LIN {X 0,Y 424.031,Z 1043.321,A -85,B 0,C 180,E1 17866.114,E2 17866.114} C_VEL
LIN {X 0,Y 429.572,Z 1017.595,A -85,B 0,C 180,E1 17864.912,E2 17864.912} C_VEL
LIN {X 0,Y 434.388,Z 990.898,A -85,B 0,C 180,E1 17863.916,E2 17863.916} C_VEL
LIN {X 0,Y 437.982,Z 968.501,A -85,B 0,C 180,E1 17863.251,E2 17863.251} C_VEL
LIN {X 0,Y 429.123,Z 944.994,A -85,B 0,C 180,E1 17861.421,E2 17861.421} C_VEL
LIN {X 0,Y 422.762,Z 922.814,A -85,B 0,C 180,E1 17859.852,E2 17859.852} C_VEL
LIN {X 0,Y 420.084,Z 910.607,A -85,B 0,C 180,E1 17859.018,E2 17859.018} C_VEL
LIN {X 0,Y 421.88,Z 885.683,A -85,B 0,C 180,E1 17856.084,E2 17856.084} C_VEL
LIN {X 0,Y 431.541,Z 834.064,A -85,B 0,C 180,E1 17850.471,E2 17850.471} C_VEL
LIN {X 0,Y 438.469,Z 800.811,A -85,B 0,C 180,E1 17846.841,E2 17846.841} C_VEL
LIN {X 0,Y 442.301,Z 782.261,A -85,B 0,C 180,E1 17844.794,E2 17844.794} C_VEL
LIN {X 0,Y 435.827,Z 764.916,A -85,B 0,C 180,E1 17841.394,E2 17841.394} C_VEL
LIN {X 0,Y 429.102,Z 747.913,A -85,B 0,C 180,E1 17837.774,E2 17837.774} C_VEL
LIN {X 0,Y 422.737,Z 732.697,A -85,B 0,C 180,E1 17834.24,E2 17834.24} C_VEL
LIN {X 0,Y 416.328,Z 717.877,A -85,B 0,C 180,E1 17830.517,E2 17830.517} C_VEL
LIN {X 0,Y 410.081,Z 704.024,A -85,B 0,C 180,E1 17826.721,E2 17826.721} C_VEL
LIN {X 0,Y 404.039,Z 691.12,A -85,B 0,C 180,E1 17822.837,E2 17822.837} C_VEL
LIN {X 0,Y 398.039,Z 678.56,A -85,B 0,C 180,E1 17818.703,E2 17818.703} C_VEL
LIN {X 0,Y 393.112,Z 668.867,A -85,B 0,C 180,E1 17815.185,E2 17815.185} C_VEL
LIN {X 0,Y 390.535,Z 663.891,A -85,B 0,C 180,E1 17813.236,E2 17813.236} C_VEL
LIN {X 0,Y 388.243,Z 659.415,A -85,B 0,C 180,E1 17811.46,E2 17811.46} C_VEL
LIN {X 0,Y 385.936,Z 654.857,A -85,B 0,C 180,E1 17809.551,E2 17809.551} C_VEL
LIN {X 0,Y 384.023,Z 650.756,A -85,B 0,C 180,E1 17807.825,E2 17807.825} C_VEL
LIN {X 0,Y 381.793,Z 647.102,A -85,B 0,C 180,E1 17806.058,E2 17806.058} C_VEL
LIN {X 0,Y 381.224,Z 645.556,A -85,B 0,C 180,E1 17805.416,E2 17805.416} C_VEL
LIN {X 0,Y 379.173,Z 642.261,A -85,B 0,C 180,E1 17803.704,E2 17803.704} C_VEL
LIN {X 0,Y 378.841,Z 640.776,A -85,B 0,C 180,E1 17803.122,E2 17803.122} C_VEL
LIN {X 0,Y 378.842,Z 640.781,A -85,B 0,C 180,E1 17799.111,E2 17799.111} C_VEL
LIN {X 0,Y 378.854,Z 640.787,A -85,B 0,C 180,E1 17795.021,E2 17795.021} C_VEL
LIN {X 0,Y 378.842,Z 640.792,A -85,B 0,C 180,E1 17790.876,E2 17790.876} C_VEL
LIN {X 0,Y 378.847,Z 640.79,A -85,B 0,C 180,E1 17786.784,E2 17786.784} C_VEL
LIN {X 0,Y 378.847,Z 640.785,A -85,B 0,C 180,E1 17782.597,E2 17782.597} C_VEL
LIN {X 0,Y 378.846,Z 640.811,A -85,B 0,C 180,E1 17781.666,E2 17781.666} C_VEL
LIN {X 0,Y 379.93,Z 643.909,A -85,B 0,C 180,E1 17781.165,E2 17781.165} C_VEL
LIN {X 0,Y 381.356,Z 646.05,A -85,B 0,C 180,E1 17780.713,E2 17780.713} C_VEL
LIN {X 0,Y 389.692,Z 662.721,A -85,B 0,C 180,E1 17777.759,E2 17777.759} C_VEL
LIN {X 0,Y 397.273,Z 679.963,A -85,B 0,C 180,E1 17774.988,E2 17774.988} C_VEL
LIN {X 0,Y 404.151,Z 697.993,A -85,B 0,C 180,E1 17772.395,E2 17772.395} C_VEL
LIN {X 0,Y 410.209,Z 717.323,A -85,B 0,C 180,E1 17769.841,E2 17769.841} C_VEL
LIN {X 0,Y 411.164,Z 721.42,A -85,B 0,C 180,E1 17769.346,E2 17769.346} C_VEL
LIN {X 0,Y 407.057,Z 767.944,A -85,B 0,C 180,E1 17765.427,E2 17765.427} C_VEL
LIN {X 0,Y 402.868,Z 818.065,A -85,B 0,C 180,E1 17761.244,E2 17761.244} C_VEL
LIN {X 0,Y 399.655,Z 864.554,A -85,B 0,C 180,E1 17757.511,E2 17757.511} C_VEL
LIN {X 0,Y 400.168,Z 872.112,A -85,B 0,C 180,E1 17757.318,E2 17757.318} C_VEL
LIN {X 0,Y 395.871,Z 1029.252,A -85,B 0,C 180,E1 17754.503,E2 17754.503} C_VEL
LIN {X 0,Y 395.432,Z 1046.821,A -85,B 0,C 180,E1 17754.006,E2 17754.006} C_VEL
LIN {X 0,Y 394.481,Z 1064.239,A -85,B 0,C 180,E1 17753.238,E2 17753.238} C_VEL
LIN {X 0,Y 393.16,Z 1080.267,A -85,B 0,C 180,E1 17752.265,E2 17752.265} C_VEL
LIN {X 0,Y 391.555,Z 1095.097,A -85,B 0,C 180,E1 17751.102,E2 17751.102} C_VEL
LIN {X 0,Y 389.588,Z 1109.913,A -85,B 0,C 180,E1 17749.623,E2 17749.623} C_VEL
LIN {X 0,Y 387.45,Z 1123.854,A -85,B 0,C 180,E1 17747.882,E2 17747.882} C_VEL
LIN {X 0,Y 385.351,Z 1136.244,A -85,B 0,C 180,E1 17745.962,E2 17745.962} C_VEL
LIN {X 0,Y 383.385,Z 1146.973,A -85,B 0,C 180,E1 17743.881,E2 17743.881} C_VEL
LIN {X 0,Y 381.545,Z 1156.777,A -85,B 0,C 180,E1 17741.486,E2 17741.486} C_VEL
LIN {X 0,Y 380.127,Z 1164.442,A -85,B 0,C 180,E1 17739.078,E2 17739.078} C_VEL
LIN {X 0,Y 379.044,Z 1170.475,A -85,B 0,C 180,E1 17736.511,E2 17736.511} C_VEL
LIN {X 0,Y 378.313,Z 1174.865,A -85,B 0,C 180,E1 17733.786,E2 17733.786} C_VEL
LIN {X 0,Y 377.955,Z 1177.371,A -85,B 0,C 180,E1 17731.059,E2 17731.059} C_VEL
LIN {X 0,Y 377.889,Z 1177.992,A -85,B 0,C 180,E1 17728.33,E2 17728.33} C_VEL
LIN {X 0,Y 378.121,Z 1176.838,A -85,B 0,C 180,E1 17725.6,E2 17725.6} C_VEL
LIN {X 0,Y 378.654,Z 1174.068,A -85,B 0,C 180,E1 17723.021,E2 17723.021} C_VEL
LIN {X 0,Y 379.541,Z 1169.524,A -85,B 0,C 180,E1 17720.444,E2 17720.444} C_VEL
LIN {X 0,Y 380.842,Z 1163.047,A -85,B 0,C 180,E1 17717.874,E2 17717.874} C_VEL
LIN {X 0,Y 382.502,Z 1155.002,A -85,B 0,C 180,E1 17715.464,E2 17715.464} C_VEL
LIN {X 0,Y 384.456,Z 1145.382,A -85,B 0,C 180,E1 17713.219,E2 17713.219} C_VEL
LIN {X 0,Y 386.621,Z 1134.139,A -85,B 0,C 180,E1 17711.137,E2 17711.137} C_VEL
LIN {X 0,Y 388.821,Z 1121.791,A -85,B 0,C 180,E1 17709.291,E2 17709.291} C_VEL
LIN {X 0,Y 390.958,Z 1108.464,A -85,B 0,C 180,E1 17707.677,E2 17707.677} C_VEL
LIN {X 0,Y 392.904,Z 1094.157,A -85,B 0,C 180,E1 17706.289,E2 17706.289} C_VEL
LIN {X 0,Y 394.624,Z 1078.729,A -85,B 0,C 180,E1 17705.107,E2 17705.107} C_VEL
LIN {X 0,Y 396.012,Z 1062.182,A -85,B 0,C 180,E1 17704.138,E2 17704.138} C_VEL
LIN {X 0,Y 396.937,Z 1045.139,A -85,B 0,C 180,E1 17703.42,E2 17703.42} C_VEL
LIN {X 0,Y 397.335,Z 1026.569,A -85,B 0,C 180,E1 17702.932,E2 17702.932} C_VEL
LIN {X 0,Y 399.086,Z 959.214,A -85,B 0,C 180,E1 17701.717,E2 17701.717} C_VEL
LIN {X 0,Y 398.467,Z 951.603,A -85,B 0,C 180,E1 17701.515,E2 17701.515} C_VEL
LIN {X 0,Y 393.586,Z 931.664,A -85,B 0,C 180,E1 17700.717,E2 17700.717} C_VEL
LIN {X 0,Y 393.131,Z 925.124,A -85,B 0,C 180,E1 17700.545,E2 17700.545} C_VEL
LIN {X 0,Y 394.72,Z 870.182,A -85,B 0,C 180,E1 17699.543,E2 17699.543} C_VEL
LIN {X 0,Y 394.254,Z 864.919,A -85,B 0,C 180,E1 17699.35,E2 17699.35} C_VEL
LIN {X 0,Y 397.972,Z 816.503,A -85,B 0,C 180,E1 17695.4,E2 17695.4} C_VEL
LIN {X 0,Y 402.393,Z 767.422,A -85,B 0,C 180,E1 17691.256,E2 17691.256} C_VEL
LIN {X 0,Y 403.838,Z 767.962,A -85,B 0,C 180,E1 17691.029,E2 17691.029} C_VEL
LIN {X 0,Y 406.516,Z 766.956,A -85,B 0,C 180,E1 17690.7,E2 17690.7} C_VEL
LIN {X 0,Y 410.432,Z 763.169,A -85,B 0,C 180,E1 17690.312,E2 17690.312} C_VEL
LIN {X 0,Y 412.105,Z 761.138,A -85,B 0,C 180,E1 17690.166,E2 17690.166} C_VEL
LIN {X 0,Y 416.175,Z 759.299,A -85,B 0,C 180,E1 17689.691,E2 17689.691} C_VEL
LIN {X 0,Y 420.888,Z 755.05,A -85,B 0,C 180,E1 17689.229,E2 17689.229} C_VEL
LIN {X 0,Y 422.259,Z 753.761,A -85,B 0,C 180,E1 17689.098,E2 17689.098} C_VEL
LIN {X 0,Y 427.431,Z 750.639,A -85,B 0,C 180,E1 17688.544,E2 17688.544} C_VEL
LIN {X 0,Y 432.452,Z 746.166,A -85,B 0,C 180,E1 17688.069,E2 17688.069} C_VEL
LIN {X 0,Y 436.101,Z 744.14,A -85,B 0,C 180,E1 17687.682,E2 17687.682} C_VEL
LIN {X 0,Y 439.705,Z 749.984,A -85,B 0,C 180,E1 17687.032,E2 17687.032} C_VEL
LIN {X 0,Y 418.06,Z 971.327,A -85,B 0,C 180,E1 17681.624,E2 17681.624} C_VEL
LIN {X 0,Y 415.617,Z 998.063,A -85,B 0,C 180,E1 17680.799,E2 17680.799} C_VEL
LIN {X 0,Y 412.746,Z 1021.843,A -85,B 0,C 180,E1 17679.809,E2 17679.809} C_VEL
LIN {X 0,Y 409.391,Z 1044.41,A -85,B 0,C 180,E1 17678.611,E2 17678.611} C_VEL
LIN {X 0,Y 405.663,Z 1065.433,A -85,B 0,C 180,E1 17677.235,E2 17677.235} C_VEL
LIN {X 0,Y 401.608,Z 1085.727,A -85,B 0,C 180,E1 17675.633,E2 17675.633} C_VEL
LIN {X 0,Y 397.135,Z 1106.048,A -85,B 0,C 180,E1 17673.726,E2 17673.726} C_VEL
LIN {X 0,Y 392.712,Z 1124.842,A -85,B 0,C 180,E1 17671.635,E2 17671.635} C_VEL
LIN {X 0,Y 388.261,Z 1142.534,A -85,B 0,C 180,E1 17669.295,E2 17669.295} C_VEL
LIN {X 0,Y 384.036,Z 1158.977,A -85,B 0,C 180,E1 17666.739,E2 17666.739} C_VEL
LIN {X 0,Y 380.255,Z 1173.722,A -85,B 0,C 180,E1 17664.053,E2 17664.053} C_VEL
LIN {X 0,Y 376.881,Z 1187.211,A -85,B 0,C 180,E1 17661.151,E2 17661.151} C_VEL
LIN {X 0,Y 374.017,Z 1199.238,A -85,B 0,C 180,E1 17658.066,E2 17658.066} C_VEL
LIN {X 0,Y 371.664,Z 1210.327,A -85,B 0,C 180,E1 17654.649,E2 17654.649} C_VEL
LIN {X 0,Y 370.099,Z 1219.053,A -85,B 0,C 180,E1 17651.375,E2 17651.375} C_VEL
LIN {X 0,Y 369.107,Z 1225.945,A -85,B 0,C 180,E1 17648.098,E2 17648.098} C_VEL
LIN {X 0,Y 368.542,Z 1231.531,A -85,B 0,C 180,E1 17644.669,E2 17644.669} C_VEL
LIN {X 0,Y 368.34,Z 1235.206,A -85,B 0,C 180,E1 17641.556,E2 17641.556} C_VEL
LIN {X 0,Y 368.303,Z 1237.705,A -85,B 0,C 180,E1 17638.133,E2 17638.133} C_VEL
LIN {X 0,Y 368.395,Z 1238.777,A -85,B 0,C 180,E1 17634.861,E2 17634.861} C_VEL
LIN {X 0,Y 368.66,Z 1238.351,A -85,B 0,C 180,E1 17631.578,E2 17631.578} C_VEL
LIN {X 0,Y 369.274,Z 1236.414,A -85,B 0,C 180,E1 17627.966,E2 17627.966} C_VEL
LIN {X 0,Y 370.42,Z 1233.083,A -85,B 0,C 180,E1 17624.5,E2 17624.5} C_VEL
LIN {X 0,Y 372.464,Z 1227.596,A -85,B 0,C 180,E1 17620.719,E2 17620.719} C_VEL
LIN {X 0,Y 375.327,Z 1220.672,A -85,B 0,C 180,E1 17617.188,E2 17617.188} C_VEL
LIN {X 0,Y 379.199,Z 1211.964,A -85,B 0,C 180,E1 17613.705,E2 17613.705} C_VEL
LIN {X 0,Y 384.057,Z 1201.512,A -85,B 0,C 180,E1 17610.352,E2 17610.352} C_VEL
LIN {X 0,Y 389.426,Z 1190.172,A -85,B 0,C 180,E1 17607.371,E2 17607.371} C_VEL
LIN {X 0,Y 395.743,Z 1176.713,A -85,B 0,C 180,E1 17604.448,E2 17604.448} C_VEL
LIN {X 0,Y 402.539,Z 1161.94,A -85,B 0,C 180,E1 17601.793,E2 17601.793} C_VEL
LIN {X 0,Y 409.684,Z 1145.817,A -85,B 0,C 180,E1 17599.381,E2 17599.381} C_VEL
LIN {X 0,Y 416.899,Z 1128.807,A -85,B 0,C 180,E1 17597.254,E2 17597.254} C_VEL
LIN {X 0,Y 424.707,Z 1109.687,A -85,B 0,C 180,E1 17595.256,E2 17595.256} C_VEL
LIN {X 0,Y 432.71,Z 1089.815,A -85,B 0,C 180,E1 17593.522,E2 17593.522} C_VEL
LIN {X 0,Y 420.838,Z 1109.322,A -85,B 0,C 180,E1 17591.796,E2 17591.796} C_VEL
LIN {X 0,Y 409.181,Z 1130.653,A -85,B 0,C 180,E1 17589.538,E2 17589.538} C_VEL
LIN {X 0,Y 398.045,Z 1155.339,A -85,B 0,C 180,E1 17586.539,E2 17586.539} C_VEL
LIN {X 0,Y 388.323,Z 1182.093,A -85,B 0,C 180,E1 17582.823,E2 17582.823} C_VEL
LIN {X 0,Y 381.527,Z 1204.921,A -85,B 0,C 180,E1 17579.176,E2 17579.176} C_VEL
LIN {X 0,Y 376.907,Z 1223.133,A -85,B 0,C 180,E1 17575.792,E2 17575.792} C_VEL
LIN {X 0,Y 373.571,Z 1238.131,A -85,B 0,C 180,E1 17572.506,E2 17572.506} C_VEL
LIN {X 0,Y 371.253,Z 1250.21,A -85,B 0,C 180,E1 17569.348,E2 17569.348} C_VEL
LIN {X 0,Y 369.717,Z 1260.007,A -85,B 0,C 180,E1 17566.241,E2 17566.241} C_VEL
LIN {X 0,Y 368.768,Z 1267.805,A -85,B 0,C 180,E1 17563.167,E2 17563.167} C_VEL
LIN {X 0,Y 368.296,Z 1273.929,A -85,B 0,C 180,E1 17560.008,E2 17560.008} C_VEL
LIN {X 0,Y 368.176,Z 1278.219,A -85,B 0,C 180,E1 17556.865,E2 17556.865} C_VEL
LIN {X 0,Y 368.227,Z 1280.634,A -85,B 0,C 180,E1 17553.895,E2 17553.895} C_VEL
LIN {X 0,Y 368.314,Z 1281.463,A -85,B 0,C 180,E1 17550.935,E2 17550.935} C_VEL
LIN {X 0,Y 368.331,Z 1280.72,A -85,B 0,C 180,E1 17547.98,E2 17547.98} C_VEL
LIN {X 0,Y 368.293,Z 1278.415,A -85,B 0,C 180,E1 17545.018,E2 17545.018} C_VEL
LIN {X 0,Y 368.285,Z 1274.288,A -85,B 0,C 180,E1 17541.886,E2 17541.886} C_VEL
LIN {X 0,Y 368.473,Z 1268.454,A -85,B 0,C 180,E1 17538.735,E2 17538.735} C_VEL
LIN {X 0,Y 369.013,Z 1260.875,A -85,B 0,C 180,E1 17535.567,E2 17535.567} C_VEL
LIN {X 0,Y 370.101,Z 1250.861,A -85,B 0,C 180,E1 17532.227,E2 17532.227} C_VEL
LIN {X 0,Y 371.775,Z 1239.387,A -85,B 0,C 180,E1 17529.043,E2 17529.043} C_VEL
LIN {X 0,Y 374.3,Z 1225.03,A -85,B 0,C 180,E1 17525.711,E2 17525.711} C_VEL
LIN {X 0,Y 377.33,Z 1209.895,A -85,B 0,C 180,E1 17522.717,E2 17522.717} C_VEL
LIN {X 0,Y 381.385,Z 1191.503,A -85,B 0,C 180,E1 17519.605,E2 17519.605} C_VEL
LIN {X 0,Y 386.238,Z 1170.811,A -85,B 0,C 180,E1 17516.628,E2 17516.628} C_VEL
LIN {X 0,Y 391.893,Z 1147.584,A -85,B 0,C 180,E1 17513.799,E2 17513.799} C_VEL
LIN {X 0,Y 397.99,Z 1122.971,A -85,B 0,C 180,E1 17511.279,E2 17511.279} C_VEL
LIN {X 0,Y 403.629,Z 1100.15,A -85,B 0,C 180,E1 17509.292,E2 17509.292} C_VEL
LIN {X 0,Y 409.926,Z 1074.472,A -85,B 0,C 180,E1 17507.403,E2 17507.403} C_VEL
LIN {X 0,Y 415.804,Z 1049.73,A -85,B 0,C 180,E1 17505.883,E2 17505.883} C_VEL
LIN {X 0,Y 421.539,Z 1023.87,A -85,B 0,C 180,E1 17504.597,E2 17504.597} C_VEL
LIN {X 0,Y 426.857,Z 997.071,A -85,B 0,C 180,E1 17503.51,E2 17503.51} C_VEL
LIN {X 0,Y 430.603,Z 975.057,A -85,B 0,C 180,E1 17502.8,E2 17502.8} C_VEL
LIN {X 0,Y 431.204,Z 970.753,A -85,B 0,C 180,E1 17502.665,E2 17502.665} C_VEL
LIN {X 0,Y 423.093,Z 948.417,A -85,B 0,C 180,E1 17500.878,E2 17500.878} C_VEL
LIN {X 0,Y 416.791,Z 926.156,A -85,B 0,C 180,E1 17499.286,E2 17499.286} C_VEL
LIN {X 0,Y 413.097,Z 908.739,A -85,B 0,C 180,E1 17498.114,E2 17498.114} C_VEL
LIN {X 0,Y 415.564,Z 883.187,A -85,B 0,C 180,E1 17495.104,E2 17495.104} C_VEL
LIN {X 0,Y 424.795,Z 836.45,A -85,B 0,C 180,E1 17489.985,E2 17489.985} C_VEL
LIN {X 0,Y 431.838,Z 803.495,A -85,B 0,C 180,E1 17486.36,E2 17486.36} C_VEL
LIN {X 0,Y 435.637,Z 785.94,A -85,B 0,C 180,E1 17484.403,E2 17484.403} C_VEL
LIN {X 0,Y 428.843,Z 767.674,A -85,B 0,C 180,E1 17480.757,E2 17480.757} C_VEL
LIN {X 0,Y 422.155,Z 750.724,A -85,B 0,C 180,E1 17477.08,E2 17477.08} C_VEL
LIN {X 0,Y 415.828,Z 735.503,A -85,B 0,C 180,E1 17473.488,E2 17473.488} C_VEL
LIN {X 0,Y 409.667,Z 721.272,A -85,B 0,C 180,E1 17469.837,E2 17469.837} C_VEL
LIN {X 0,Y 403.651,Z 708.035,A -85,B 0,C 180,E1 17466.115,E2 17466.115} C_VEL
LIN {X 0,Y 398.299,Z 696.472,A -85,B 0,C 180,E1 17462.59,E2 17462.59} C_VEL
LIN {X 0,Y 392.484,Z 684.232,A -85,B 0,C 180,E1 17458.54,E2 17458.54} C_VEL
LIN {X 0,Y 387.464,Z 674.344,A -85,B 0,C 180,E1 17454.913,E2 17454.913} C_VEL
LIN {X 0,Y 384.753,Z 669.087,A -85,B 0,C 180,E1 17452.834,E2 17452.834} C_VEL
LIN {X 0,Y 382.847,Z 665.228,A -85,B 0,C 180,E1 17451.287,E2 17451.287} C_VEL
LIN {X 0,Y 380.499,Z 660.623,A -85,B 0,C 180,E1 17449.346,E2 17449.346} C_VEL
LIN {X 0,Y 378.183,Z 656.035,A -85,B 0,C 180,E1 17447.307,E2 17447.307} C_VEL
LIN {X 0,Y 376.218,Z 652.07,A -85,B 0,C 180,E1 17445.533,E2 17445.533} C_VEL
LIN {X 0,Y 373.885,Z 648.166,A -85,B 0,C 180,E1 17443.532,E2 17443.532} C_VEL
LIN {X 0,Y 373.366,Z 646.607,A -85,B 0,C 180,E1 17442.867,E2 17442.867} C_VEL
LIN {X 0,Y 371.234,Z 643.221,A -85,B 0,C 180,E1 17440.968,E2 17440.968} C_VEL
LIN {X 0,Y 370.909,Z 641.765,A -85,B 0,C 180,E1 17440.307,E2 17440.307} C_VEL
LIN {X 0,Y 370.904,Z 641.763,A -85,B 0,C 180,E1 17436.317,E2 17436.317} C_VEL
LIN {X 0,Y 370.921,Z 641.762,A -85,B 0,C 180,E1 17432.146,E2 17432.146} C_VEL
LIN {X 0,Y 370.904,Z 641.769,A -85,B 0,C 180,E1 17427.922,E2 17427.922} C_VEL
LIN {X 0,Y 370.903,Z 641.77,A -85,B 0,C 180,E1 17423.815,E2 17423.815} C_VEL
LIN {X 0,Y 370.931,Z 641.954,A -85,B 0,C 180,E1 17422.896,E2 17422.896} C_VEL
LIN {X 0,Y 371.968,Z 644.859,A -85,B 0,C 180,E1 17422.396,E2 17422.396} C_VEL
LIN {X 0,Y 373.417,Z 646.919,A -85,B 0,C 180,E1 17421.924,E2 17421.924} C_VEL
LIN {X 0,Y 375.245,Z 650.541,A -85,B 0,C 180,E1 17421.23,E2 17421.23} C_VEL
LIN {X 0,Y 382.114,Z 664.007,A -85,B 0,C 180,E1 17418.744,E2 17418.744} C_VEL
LIN {X 0,Y 389.704,Z 680.901,A -85,B 0,C 180,E1 17415.92,E2 17415.92} C_VEL
LIN {X 0,Y 396.49,Z 698.381,A -85,B 0,C 180,E1 17413.306,E2 17413.306} C_VEL
LIN {X 0,Y 402.531,Z 717.046,A -85,B 0,C 180,E1 17410.744,E2 17410.744} C_VEL
LIN {X 0,Y 404.439,Z 724.573,A -85,B 0,C 180,E1 17409.813,E2 17409.813} C_VEL
LIN {X 0,Y 399.978,Z 772.795,A -85,B 0,C 180,E1 17405.709,E2 17405.709} C_VEL
LIN {X 0,Y 395.761,Z 821.856,A -85,B 0,C 180,E1 17401.59,E2 17401.59} C_VEL
LIN {X 0,Y 392.655,Z 865.628,A -85,B 0,C 180,E1 17398.053,E2 17398.053} C_VEL
LIN {X 0,Y 393.135,Z 872.997,A -85,B 0,C 180,E1 17397.862,E2 17397.862} C_VEL
LIN {X 0,Y 388.676,Z 1029.669,A -85,B 0,C 180,E1 17395.01,E2 17395.01} C_VEL
LIN {X 0,Y 388.231,Z 1047.32,A -85,B 0,C 180,E1 17394.51,E2 17394.51} C_VEL
LIN {X 0,Y 387.271,Z 1064.483,A -85,B 0,C 180,E1 17393.749,E2 17393.749} C_VEL
LIN {X 0,Y 385.935,Z 1080.296,A -85,B 0,C 180,E1 17392.786,E2 17392.786} C_VEL
LIN {X 0,Y 384.167,Z 1096.172,A -85,B 0,C 180,E1 17391.527,E2 17391.527} C_VEL
LIN {X 0,Y 382.153,Z 1110.788,A -85,B 0,C 180,E1 17390.042,E2 17390.042} C_VEL
LIN {X 0,Y 379.908,Z 1124.888,A -85,B 0,C 180,E1 17388.25,E2 17388.25} C_VEL
LIN {X 0,Y 377.728,Z 1137.262,A -85,B 0,C 180,E1 17386.293,E2 17386.293} C_VEL
LIN {X 0,Y 375.683,Z 1147.979,A -85,B 0,C 180,E1 17384.171,E2 17384.171} C_VEL
LIN {X 0,Y 373.766,Z 1157.774,A -85,B 0,C 180,E1 17381.728,E2 17381.728} C_VEL
LIN {X 0,Y 372.286,Z 1165.429,A -85,B 0,C 180,E1 17379.271,E2 17379.271} C_VEL
LIN {X 0,Y 371.154,Z 1171.452,A -85,B 0,C 180,E1 17376.65,E2 17376.65} C_VEL
LIN {X 0,Y 370.389,Z 1175.834,A -85,B 0,C 180,E1 17373.868,E2 17373.868} C_VEL
LIN {X 0,Y 370.015,Z 1178.33,A -85,B 0,C 180,E1 17371.082,E2 17371.082} C_VEL
LIN {X 0,Y 369.947,Z 1178.944,A -85,B 0,C 180,E1 17368.294,E2 17368.294} C_VEL
LIN {X 0,Y 370.194,Z 1177.782,A -85,B 0,C 180,E1 17365.505,E2 17365.505} C_VEL
LIN {X 0,Y 370.758,Z 1175.005,A -85,B 0,C 180,E1 17362.872,E2 17362.872} C_VEL
LIN {X 0,Y 371.692,Z 1170.449,A -85,B 0,C 180,E1 17360.241,E2 17360.241} C_VEL
LIN {X 0,Y 373.06,Z 1163.964,A -85,B 0,C 180,E1 17357.617,E2 17357.617} C_VEL
LIN {X 0,Y 374.798,Z 1155.909,A -85,B 0,C 180,E1 17355.159,E2 17355.159} C_VEL
LIN {X 0,Y 376.839,Z 1146.271,A -85,B 0,C 180,E1 17352.869,E2 17352.869} C_VEL
LIN {X 0,Y 379.095,Z 1135.014,A -85,B 0,C 180,E1 17350.748,E2 17350.748} C_VEL
LIN {X 0,Y 381.386,Z 1122.649,A -85,B 0,C 180,E1 17348.868,E2 17348.868} C_VEL
LIN {X 0,Y 383.606,Z 1109.298,A -85,B 0,C 180,E1 17347.226,E2 17347.226} C_VEL
LIN {X 0,Y 385.627,Z 1094.952,A -85,B 0,C 180,E1 17345.814,E2 17345.814} C_VEL
LIN {X 0,Y 387.447,Z 1079.156,A -85,B 0,C 180,E1 17344.589,E2 17344.589} C_VEL
LIN {X 0,Y 388.855,Z 1062.87,A -85,B 0,C 180,E1 17343.626,E2 17343.626} C_VEL
LIN {X 0,Y 389.807,Z 1045.815,A -85,B 0,C 180,E1 17342.9,E2 17342.9} C_VEL
LIN {X 0,Y 390.222,Z 1027.284,A -85,B 0,C 180,E1 17342.408,E2 17342.408} C_VEL
LIN {X 0,Y 393.131,Z 925.124,A -85,B 0,C 180,E1 17340.545,E2 17340.545} C_VEL
LIN {X 0,Y 392.509,Z 917.516,A -85,B 0,C 180,E1 17340.336,E2 17340.336} C_VEL
LIN {X 0,Y 387.765,Z 897.575,A -85,B 0,C 180,E1 17339.513,E2 17339.513} C_VEL
LIN {X 0,Y 387.342,Z 891.036,A -85,B 0,C 180,E1 17339.338,E2 17339.338} C_VEL
LIN {X 0,Y 387.821,Z 871.104,A -85,B 0,C 180,E1 17338.958,E2 17338.958} C_VEL
LIN {X 0,Y 387.337,Z 866.12,A -85,B 0,C 180,E1 17338.785,E2 17338.785} C_VEL
LIN {X 0,Y 391.297,Z 816.823,A -85,B 0,C 180,E1 17334.723,E2 17334.723} C_VEL
LIN {X 0,Y 394.531,Z 781.853,A -85,B 0,C 180,E1 17331.754,E2 17331.754} C_VEL
LIN {X 0,Y 396.413,Z 782.323,A -85,B 0,C 180,E1 17331.461,E2 17331.461} C_VEL
LIN {X 0,Y 399.357,Z 780.833,A -85,B 0,C 180,E1 17331.109,E2 17331.109} C_VEL
LIN {X 0,Y 403.511,Z 776.395,A -85,B 0,C 180,E1 17330.717,E2 17330.717} C_VEL
LIN {X 0,Y 404.367,Z 775.584,A -85,B 0,C 180,E1 17330.633,E2 17330.633} C_VEL
LIN {X 0,Y 408.466,Z 773.667,A -85,B 0,C 180,E1 17330.151,E2 17330.151} C_VEL
LIN {X 0,Y 413.122,Z 769.361,A -85,B 0,C 180,E1 17329.695,E2 17329.695} C_VEL
LIN {X 0,Y 414.607,Z 767.993,A -85,B 0,C 180,E1 17329.552,E2 17329.552} C_VEL
LIN {X 0,Y 419.822,Z 764.787,A -85,B 0,C 180,E1 17328.991,E2 17328.991} C_VEL
LIN {X 0,Y 424.467,Z 760.542,A -85,B 0,C 180,E1 17328.551,E2 17328.551} C_VEL
LIN {X 0,Y 430.338,Z 756.683,A -85,B 0,C 180,E1 17327.951,E2 17327.951} C_VEL
LIN {X 0,Y 433.438,Z 754.075,A -85,B 0,C 180,E1 17327.656,E2 17327.656} C_VEL
LIN {X 0,Y 413.612,Z 946.997,A -85,B 0,C 180,E1 17322.884,E2 17322.884} C_VEL
LIN {X 0,Y 409.476,Z 992.588,A -85,B 0,C 180,E1 17321.596,E2 17321.596} C_VEL
LIN {X 0,Y 406.679,Z 1016.293,A -85,B 0,C 180,E1 17320.659,E2 17320.659} C_VEL
LIN {X 0,Y 403.374,Z 1038.862,A -85,B 0,C 180,E1 17319.507,E2 17319.507} C_VEL
LIN {X 0,Y 399.41,Z 1061.529,A -85,B 0,C 180,E1 17318.074,E2 17318.074} C_VEL
LIN {X 0,Y 395.281,Z 1082.349,A -85,B 0,C 180,E1 17316.474,E2 17316.474} C_VEL
LIN {X 0,Y 390.795,Z 1102.55,A -85,B 0,C 180,E1 17314.612,E2 17314.612} C_VEL
LIN {X 0,Y 386.307,Z 1121.144,A -85,B 0,C 180,E1 17312.573,E2 17312.573} C_VEL
LIN {X 0,Y 381.549,Z 1139.942,A -85,B 0,C 180,E1 17310.138,E2 17310.138} C_VEL
LIN {X 0,Y 377.256,Z 1156.35,A -85,B 0,C 180,E1 17307.634,E2 17307.634} C_VEL
LIN {X 0,Y 373.215,Z 1171.649,A -85,B 0,C 180,E1 17304.874,E2 17304.874} C_VEL
LIN {X 0,Y 369.615,Z 1185.489,A -85,B 0,C 180,E1 17301.921,E2 17301.921} C_VEL
LIN {X 0,Y 366.564,Z 1197.932,A -85,B 0,C 180,E1 17298.776,E2 17298.776} C_VEL
LIN {X 0,Y 364.224,Z 1208.457,A -85,B 0,C 180,E1 17295.607,E2 17295.607} C_VEL
LIN {X 0,Y 362.449,Z 1217.529,A -85,B 0,C 180,E1 17292.264,E2 17292.264} C_VEL
LIN {X 0,Y 361.27,Z 1225.221,A -85,B 0,C 180,E1 17288.756,E2 17288.756} C_VEL
LIN {X 0,Y 360.643,Z 1230.954,A -85,B 0,C 180,E1 17285.409,E2 17285.409} C_VEL
LIN {X 0,Y 360.364,Z 1235.075,A -85,B 0,C 180,E1 17282.067,E2 17282.067} C_VEL
LIN {X 0,Y 360.314,Z 1237.87,A -85,B 0,C 180,E1 17278.728,E2 17278.728} C_VEL
LIN {X 0,Y 360.381,Z 1239.171,A -85,B 0,C 180,E1 17275.385,E2 17275.385} C_VEL
LIN {X 0,Y 360.668,Z 1239.116,A -85,B 0,C 180,E1 17271.786,E2 17271.786} C_VEL
LIN {X 0,Y 361.274,Z 1237.568,A -85,B 0,C 180,E1 17268.182,E2 17268.182} C_VEL
LIN {X 0,Y 362.489,Z 1234.288,A -85,B 0,C 180,E1 17264.481,E2 17264.481} C_VEL
LIN {X 0,Y 364.507,Z 1229.362,A -85,B 0,C 180,E1 17260.781,E2 17260.781} C_VEL
LIN {X 0,Y 367.673,Z 1222.387,A -85,B 0,C 180,E1 17256.945,E2 17256.945} C_VEL
LIN {X 0,Y 371.633,Z 1214.229,A -85,B 0,C 180,E1 17253.472,E2 17253.472} C_VEL
LIN {X 0,Y 376.446,Z 1204.749,A -85,B 0,C 180,E1 17250.218,E2 17250.218} C_VEL
LIN {X 0,Y 382.577,Z 1192.764,A -85,B 0,C 180,E1 17246.891,E2 17246.891} C_VEL
LIN {X 0,Y 389.495,Z 1179.159,A -85,B 0,C 180,E1 17243.811,E2 17243.811} C_VEL
LIN {X 0,Y 397.083,Z 1163.924,A -85,B 0,C 180,E1 17240.985,E2 17240.985} C_VEL
LIN {X 0,Y 404.743,Z 1148.035,A -85,B 0,C 180,E1 17238.541,E2 17238.541} C_VEL
LIN {X 0,Y 413,Z 1130.334,A -85,B 0,C 180,E1 17236.274,E2 17236.274} C_VEL
LIN {X 0,Y 422.364,Z 1109.922,A -85,B 0,C 180,E1 17234.109,E2 17234.109} C_VEL
LIN {X 0,Y 424.839,Z 1104.283,A -85,B 0,C 180,E1 17233.553,E2 17233.553} C_VEL
LIN {X 0,Y 412.217,Z 1123.286,A -85,B 0,C 180,E1 17231.655,E2 17231.655} C_VEL
LIN {X 0,Y 400.152,Z 1143.996,A -85,B 0,C 180,E1 17229.214,E2 17229.214} C_VEL
LIN {X 0,Y 388.536,Z 1168.241,A -85,B 0,C 180,E1 17225.929,E2 17225.929} C_VEL
LIN {X 0,Y 378.618,Z 1194.364,A -85,B 0,C 180,E1 17221.884,E2 17221.884} C_VEL
LIN {X 0,Y 372.234,Z 1214.763,A -85,B 0,C 180,E1 17218.216,E2 17218.216} C_VEL
LIN {X 0,Y 367.836,Z 1231.23,A -85,B 0,C 180,E1 17214.749,E2 17214.749} C_VEL
LIN {X 0,Y 364.84,Z 1244.153,A -85,B 0,C 180,E1 17211.548,E2 17211.548} C_VEL
LIN {X 0,Y 362.608,Z 1255.53,A -85,B 0,C 180,E1 17208.157,E2 17208.157} C_VEL
LIN {X 0,Y 361.241,Z 1264.327,A -85,B 0,C 180,E1 17204.919,E2 17204.919} C_VEL
LIN {X 0,Y 360.491,Z 1271.192,A -85,B 0,C 180,E1 17201.684,E2 17201.684} C_VEL
LIN {X 0,Y 360.205,Z 1276.207,A -85,B 0,C 180,E1 17198.462,E2 17198.462} C_VEL
LIN {X 0,Y 360.196,Z 1279.286,A -85,B 0,C 180,E1 17195.418,E2 17195.418} C_VEL
LIN {X 0,Y 360.287,Z 1280.758,A -85,B 0,C 180,E1 17192.388,E2 17192.388} C_VEL
LIN {X 0,Y 360.355,Z 1280.643,A -85,B 0,C 180,E1 17189.366,E2 17189.366} C_VEL
LIN {X 0,Y 360.336,Z 1278.963,A -85,B 0,C 180,E1 17186.343,E2 17186.343} C_VEL
LIN {X 0,Y 360.298,Z 1275.72,A -85,B 0,C 180,E1 17183.309,E2 17183.309} C_VEL
LIN {X 0,Y 360.383,Z 1270.541,A -85,B 0,C 180,E1 17180.051,E2 17180.051} C_VEL
LIN {X 0,Y 360.749,Z 1263.783,A -85,B 0,C 180,E1 17176.865,E2 17176.865} C_VEL
LIN {X 0,Y 361.575,Z 1255.072,A -85,B 0,C 180,E1 17173.619,E2 17173.619} C_VEL
LIN {X 0,Y 363.068,Z 1243.91,A -85,B 0,C 180,E1 17170.202,E2 17170.202} C_VEL
LIN {X 0,Y 365.236,Z 1230.949,A -85,B 0,C 180,E1 17166.905,E2 17166.905} C_VEL
LIN {X 0,Y 368.172,Z 1215.957,A -85,B 0,C 180,E1 17163.667,E2 17163.667} C_VEL
LIN {X 0,Y 372.108,Z 1197.967,A -85,B 0,C 180,E1 17160.371,E2 17160.371} C_VEL
LIN {X 0,Y 376.898,Z 1177.756,A -85,B 0,C 180,E1 17157.238,E2 17157.238} C_VEL
LIN {X 0,Y 382.202,Z 1156.322,A -85,B 0,C 180,E1 17154.415,E2 17154.415} C_VEL
LIN {X 0,Y 387.725,Z 1134.365,A -85,B 0,C 180,E1 17151.953,E2 17151.953} C_VEL
LIN {X 0,Y 393.451,Z 1112.043,A -85,B 0,C 180,E1 17149.8,E2 17149.8} C_VEL
LIN {X 0,Y 399.741,Z 1087.149,A -85,B 0,C 180,E1 17147.766,E2 17147.766} C_VEL
LIN {X 0,Y 405.799,Z 1062.879,A -85,B 0,C 180,E1 17146.086,E2 17146.086} C_VEL
LIN {X 0,Y 411.795,Z 1037.515,A -85,B 0,C 180,E1 17144.651,E2 17144.651} C_VEL
LIN {X 0,Y 418.027,Z 1009.204,A -85,B 0,C 180,E1 17143.353,E2 17143.353} C_VEL
LIN {X 0,Y 423.019,Z 982.138,A -85,B 0,C 180,E1 17142.347,E2 17142.347} C_VEL
LIN {X 0,Y 424.459,Z 973.014,A -85,B 0,C 180,E1 17142.072,E2 17142.072} C_VEL
LIN {X 0,Y 417.259,Z 952.685,A -85,B 0,C 180,E1 17140.407,E2 17140.407} C_VEL
LIN {X 0,Y 410.942,Z 929.868,A -85,B 0,C 180,E1 17138.728,E2 17138.728} C_VEL
LIN {X 0,Y 406.298,Z 907.138,A -85,B 0,C 180,E1 17137.202,E2 17137.202} C_VEL
LIN {X 0,Y 409.097,Z 882.426,A -85,B 0,C 180,E1 17134.302,E2 17134.302} C_VEL
LIN {X 0,Y 418.081,Z 838.836,A -85,B 0,C 180,E1 17129.483,E2 17129.483} C_VEL
LIN {X 0,Y 425.41,Z 805.389,A -85,B 0,C 180,E1 17125.774,E2 17125.774} C_VEL
LIN {X 0,Y 428.917,Z 789.433,A -85,B 0,C 180,E1 17123.966,E2 17123.966} C_VEL
LIN {X 0,Y 422.062,Z 770.984,A -85,B 0,C 180,E1 17120.236,E2 17120.236} C_VEL
LIN {X 0,Y 415.642,Z 754.638,A -85,B 0,C 180,E1 17116.635,E2 17116.635} C_VEL
LIN {X 0,Y 409.333,Z 739.45,A -85,B 0,C 180,E1 17112.987,E2 17112.987} C_VEL
LIN {X 0,Y 403.446,Z 725.745,A -85,B 0,C 180,E1 17109.414,E2 17109.414} C_VEL
LIN {X 0,Y 397.692,Z 712.969,A -85,B 0,C 180,E1 17105.772,E2 17105.772} C_VEL
LIN {X 0,Y 392.539,Z 701.791,A -85,B 0,C 180,E1 17102.336,E2 17102.336} C_VEL
LIN {X 0,Y 386.923,Z 689.888,A -85,B 0,C 180,E1 17098.371,E2 17098.371} C_VEL
LIN {X 0,Y 381.999,Z 680.08,A -85,B 0,C 180,E1 17094.744,E2 17094.744} C_VEL
LIN {X 0,Y 378.991,Z 674.236,A -85,B 0,C 180,E1 17092.42,E2 17092.42} C_VEL
LIN {X 0,Y 377.459,Z 671.051,A -85,B 0,C 180,E1 17091.125,E2 17091.125} C_VEL
LIN {X 0,Y 374.996,Z 666.28,A -85,B 0,C 180,E1 17089.087,E2 17089.087} C_VEL
LIN {X 0,Y 372.824,Z 661.904,A -85,B 0,C 180,E1 17087.138,E2 17087.138} C_VEL
LIN {X 0,Y 370.455,Z 657.276,A -85,B 0,C 180,E1 17084.983,E2 17084.983} C_VEL
LIN {X 0,Y 368.425,Z 653.503,A -85,B 0,C 180,E1 17083.118,E2 17083.118} C_VEL
LIN {X 0,Y 367.703,Z 652.186,A -85,B 0,C 180,E1 17082.432,E2 17082.432} C_VEL
LIN {X 0,Y 365.814,Z 648.596,A -85,B 0,C 180,E1 17080.552,E2 17080.552} C_VEL
LIN {X 0,Y 365.191,Z 647.358,A -85,B 0,C 180,E1 17079.898,E2 17079.898} C_VEL
LIN {X 0,Y 363.281,Z 644.195,A -85,B 0,C 180,E1 17078.017,E2 17078.017} C_VEL
LIN {X 0,Y 362.965,Z 642.758,A -85,B 0,C 180,E1 17077.315,E2 17077.315} C_VEL
LIN {X 0,Y 362.966,Z 642.751,A -85,B 0,C 180,E1 17073.189,E2 17073.189} C_VEL
LIN {X 0,Y 362.972,Z 642.748,A -85,B 0,C 180,E1 17068.993,E2 17068.993} C_VEL
LIN {X 0,Y 362.962,Z 642.748,A -85,B 0,C 180,E1 17064.847,E2 17064.847} C_VEL
LIN {X 0,Y 362.995,Z 642.975,A -85,B 0,C 180,E1 17064.229,E2 17064.229} C_VEL
LIN {X 0,Y 364.243,Z 646.206,A -85,B 0,C 180,E1 17063.633,E2 17063.633} C_VEL
LIN {X 0,Y 365.577,Z 647.899,A -85,B 0,C 180,E1 17063.202,E2 17063.202} C_VEL
LIN {X 0,Y 367.47,Z 651.68,A -85,B 0,C 180,E1 17062.446,E2 17062.446} C_VEL
LIN {X 0,Y 374.444,Z 665.008,A -85,B 0,C 180,E1 17059.843,E2 17059.843} C_VEL
LIN {X 0,Y 382.472,Z 682.621,A -85,B 0,C 180,E1 17056.769,E2 17056.769} C_VEL
LIN {X 0,Y 389.421,Z 700.31,A -85,B 0,C 180,E1 17054.033,E2 17054.033} C_VEL
LIN {X 0,Y 395.056,Z 717.528,A -85,B 0,C 180,E1 17051.59,E2 17051.59} C_VEL
LIN {X 0,Y 397.699,Z 727.362,A -85,B 0,C 180,E1 17050.309,E2 17050.309} C_VEL
LIN {X 0,Y 393.368,Z 773.02,A -85,B 0,C 180,E1 17046.405,E2 17046.405} C_VEL
LIN {X 0,Y 388.985,Z 822.02,A -85,B 0,C 180,E1 17042.253,E2 17042.253} C_VEL
LIN {X 0,Y 385.685,Z 866.629,A -85,B 0,C 180,E1 17038.617,E2 17038.617} C_VEL
LIN {X 0,Y 386.139,Z 873.877,A -85,B 0,C 180,E1 17038.425,E2 17038.425} C_VEL
LIN {X 0,Y 381.514,Z 1029.966,A -85,B 0,C 180,E1 17035.539,E2 17035.539} C_VEL
LIN {X 0,Y 381.063,Z 1047.819,A -85,B 0,C 180,E1 17035.034,E2 17035.034} C_VEL
LIN {X 0,Y 380.073,Z 1064.989,A -85,B 0,C 180,E1 17034.266,E2 17034.266} C_VEL
LIN {X 0,Y 378.626,Z 1081.516,A -85,B 0,C 180,E1 17033.243,E2 17033.243} C_VEL
LIN {X 0,Y 376.802,Z 1097.246,A -85,B 0,C 180,E1 17031.97,E2 17031.97} C_VEL
LIN {X 0,Y 374.712,Z 1111.837,A -85,B 0,C 180,E1 17030.458,E2 17030.458} C_VEL
LIN {X 0,Y 372.382,Z 1125.922,A -85,B 0,C 180,E1 17028.632,E2 17028.632} C_VEL
LIN {X 0,Y 370.118,Z 1138.28,A -85,B 0,C 180,E1 17026.638,E2 17026.638} C_VEL
LIN {X 0,Y 367.992,Z 1148.984,A -85,B 0,C 180,E1 17024.474,E2 17024.474} C_VEL
LIN {X 0,Y 365.995,Z 1158.771,A -85,B 0,C 180,E1 17021.981,E2 17021.981} C_VEL
LIN {X 0,Y 364.451,Z 1166.415,A -85,B 0,C 180,E1 17019.472,E2 17019.472} C_VEL
LIN {X 0,Y 363.267,Z 1172.429,A -85,B 0,C 180,E1 17016.795,E2 17016.795} C_VEL
LIN {X 0,Y 362.466,Z 1176.803,A -85,B 0,C 180,E1 17013.952,E2 17013.952} C_VEL
LIN {X 0,Y 362.074,Z 1179.289,A -85,B 0,C 180,E1 17011.105,E2 17011.105} C_VEL
LIN {X 0,Y 362.006,Z 1179.895,A -85,B 0,C 180,E1 17008.257,E2 17008.257} C_VEL
LIN {X 0,Y 362.268,Z 1178.726,A -85,B 0,C 180,E1 17005.407,E2 17005.407} C_VEL
LIN {X 0,Y 362.864,Z 1175.943,A -85,B 0,C 180,E1 17002.716,E2 17002.716} C_VEL
LIN {X 0,Y 363.848,Z 1171.375,A -85,B 0,C 180,E1 17000.028,E2 17000.028} C_VEL
LIN {X 0,Y 365.285,Z 1164.88,A -85,B 0,C 180,E1 16997.349,E2 16997.349} C_VEL
LIN {X 0,Y 367.105,Z 1156.815,A -85,B 0,C 180,E1 16994.84,E2 16994.84} C_VEL
LIN {X 0,Y 369.235,Z 1147.16,A -85,B 0,C 180,E1 16992.505,E2 16992.505} C_VEL
LIN {X 0,Y 371.587,Z 1135.889,A -85,B 0,C 180,E1 16990.343,E2 16990.343} C_VEL
LIN {X 0,Y 373.971,Z 1123.506,A -85,B 0,C 180,E1 16988.428,E2 16988.428} C_VEL
LIN {X 0,Y 376.279,Z 1110.13,A -85,B 0,C 180,E1 16986.756,E2 16986.756} C_VEL
LIN {X 0,Y 378.378,Z 1095.747,A -85,B 0,C 180,E1 16985.32,E2 16985.32} C_VEL
LIN {X 0,Y 380.303,Z 1079.578,A -85,B 0,C 180,E1 16984.052,E2 16984.052} C_VEL
LIN {X 0,Y 381.788,Z 1062.851,A -85,B 0,C 180,E1 16983.057,E2 16983.057} C_VEL
LIN {X 0,Y 382.736,Z 1045.741,A -85,B 0,C 180,E1 16982.337,E2 16982.337} C_VEL
LIN {X 0,Y 383.157,Z 1026.651,A -85,B 0,C 180,E1 16981.837,E2 16981.837} C_VEL
LIN {X 0,Y 387.342,Z 891.036,A -85,B 0,C 180,E1 16979.338,E2 16979.338} C_VEL
LIN {X 0,Y 386.699,Z 886.01,A -85,B 0,C 180,E1 16979.174,E2 16979.174} C_VEL
LIN {X 0,Y 381.208,Z 872.033,A -85,B 0,C 180,E1 16978.374,E2 16978.374} C_VEL
LIN {X 0,Y 380.655,Z 869.149,A -85,B 0,C 180,E1 16978.26,E2 16978.26} C_VEL
LIN {X 0,Y 380.54,Z 866.381,A -85,B 0,C 180,E1 16978.118,E2 16978.118} C_VEL
LIN {X 0,Y 384.589,Z 818.117,A -85,B 0,C 180,E1 16974.105,E2 16974.105} C_VEL
LIN {X 0,Y 386.782,Z 796.41,A -85,B 0,C 180,E1 16972.215,E2 16972.215} C_VEL
LIN {X 0,Y 388.899,Z 796.629,A -85,B 0,C 180,E1 16971.897,E2 16971.897} C_VEL
LIN {X 0,Y 392.139,Z 794.633,A -85,B 0,C 180,E1 16971.524,E2 16971.524} C_VEL
LIN {X 0,Y 396.171,Z 790.034,A -85,B 0,C 180,E1 16971.155,E2 16971.155} C_VEL
LIN {X 0,Y 400.261,Z 788.266,A -85,B 0,C 180,E1 16970.66,E2 16970.66} C_VEL
LIN {X 0,Y 404.835,Z 784.257,A -85,B 0,C 180,E1 16970.206,E2 16970.206} C_VEL
LIN {X 0,Y 406.466,Z 782.576,A -85,B 0,C 180,E1 16970.053,E2 16970.053} C_VEL
LIN {X 0,Y 411.49,Z 779.609,A -85,B 0,C 180,E1 16969.501,E2 16969.501} C_VEL
LIN {X 0,Y 417.013,Z 774.661,A -85,B 0,C 180,E1 16968.974,E2 16968.974} C_VEL
LIN {X 0,Y 422.922,Z 770.649,A -85,B 0,C 180,E1 16968.366,E2 16968.366} C_VEL
LIN {X 0,Y 426.136,Z 767.831,A -85,B 0,C 180,E1 16968.065,E2 16968.065} C_VEL
LIN {X 0,Y 406.272,Z 954.541,A -85,B 0,C 180,E1 16963.318,E2 16963.318} C_VEL
LIN {X 0,Y 402.47,Z 994.917,A -85,B 0,C 180,E1 16962.122,E2 16962.122} C_VEL
LIN {X 0,Y 399.678,Z 1017.784,A -85,B 0,C 180,E1 16961.192,E2 16961.192} C_VEL
LIN {X 0,Y 396.339,Z 1039.888,A -85,B 0,C 180,E1 16960.04,E2 16960.04} C_VEL
LIN {X 0,Y 392.21,Z 1062.833,A -85,B 0,C 180,E1 16958.559,E2 16958.559} C_VEL
LIN {X 0,Y 387.922,Z 1083.803,A -85,B 0,C 180,E1 16956.911,E2 16956.911} C_VEL
LIN {X 0,Y 383.292,Z 1104.079,A -85,B 0,C 180,E1 16955,E2 16955} C_VEL
LIN {X 0,Y 378.616,Z 1122.915,A -85,B 0,C 180,E1 16952.878,E2 16952.878} C_VEL
LIN {X 0,Y 373.881,Z 1141.088,A -85,B 0,C 180,E1 16950.462,E2 16950.462} C_VEL
LIN {X 0,Y 369.502,Z 1157.402,A -85,B 0,C 180,E1 16947.914,E2 16947.914} C_VEL
LIN {X 0,Y 365.375,Z 1172.657,A -85,B 0,C 180,E1 16945.099,E2 16945.099} C_VEL
LIN {X 0,Y 361.702,Z 1186.437,A -85,B 0,C 180,E1 16942.084,E2 16942.084} C_VEL
LIN {X 0,Y 358.454,Z 1199.383,A -85,B 0,C 180,E1 16938.711,E2 16938.711} C_VEL
LIN {X 0,Y 356.115,Z 1209.787,A -85,B 0,C 180,E1 16935.47,E2 16935.47} C_VEL
LIN {X 0,Y 354.357,Z 1218.738,A -85,B 0,C 180,E1 16932.052,E2 16932.052} C_VEL
LIN {X 0,Y 353.203,Z 1226.278,A -85,B 0,C 180,E1 16928.465,E2 16928.465} C_VEL
LIN {X 0,Y 352.602,Z 1231.909,A -85,B 0,C 180,E1 16925.043,E2 16925.043} C_VEL
LIN {X 0,Y 352.359,Z 1235.917,A -85,B 0,C 180,E1 16921.626,E2 16921.626} C_VEL
LIN {X 0,Y 352.328,Z 1238.655,A -85,B 0,C 180,E1 16918.048,E2 16918.048} C_VEL
LIN {X 0,Y 352.435,Z 1239.827,A -85,B 0,C 180,E1 16914.774,E2 16914.774} C_VEL
LIN {X 0,Y 352.756,Z 1239.673,A -85,B 0,C 180,E1 16911.195,E2 16911.195} C_VEL
LIN {X 0,Y 353.473,Z 1238.116,A -85,B 0,C 180,E1 16907.585,E2 16907.585} C_VEL
LIN {X 0,Y 354.863,Z 1234.857,A -85,B 0,C 180,E1 16903.802,E2 16903.802} C_VEL
LIN {X 0,Y 357.127,Z 1229.932,A -85,B 0,C 180,E1 16900.027,E2 16900.027} C_VEL
LIN {X 0,Y 360.477,Z 1223.264,A -85,B 0,C 180,E1 16896.259,E2 16896.259} C_VEL
LIN {X 0,Y 364.954,Z 1214.856,A -85,B 0,C 180,E1 16892.587,E2 16892.587} C_VEL
LIN {X 0,Y 370.407,Z 1204.943,A -85,B 0,C 180,E1 16889.142,E2 16889.142} C_VEL
LIN {X 0,Y 376.726,Z 1193.619,A -85,B 0,C 180,E1 16885.942,E2 16885.942} C_VEL
LIN {X 0,Y 384.114,Z 1180.219,A -85,B 0,C 180,E1 16882.849,E2 16882.849} C_VEL
LIN {X 0,Y 392.194,Z 1165.305,A -85,B 0,C 180,E1 16880.024,E2 16880.024} C_VEL
LIN {X 0,Y 400.798,Z 1148.942,A -85,B 0,C 180,E1 16877.462,E2 16877.462} C_VEL
LIN {X 0,Y 410.701,Z 1129.762,A -85,B 0,C 180,E1 16874.988,E2 16874.988} C_VEL
LIN {X 0,Y 417.009,Z 1117.356,A -85,B 0,C 180,E1 16873.616,E2 16873.616} C_VEL
LIN {X 0,Y 403.208,Z 1136.644,A -85,B 0,C 180,E1 16871.463,E2 16871.463} C_VEL
LIN {X 0,Y 391.342,Z 1155.862,A -85,B 0,C 180,E1 16868.944,E2 16868.944} C_VEL
LIN {X 0,Y 380.228,Z 1177.478,A -85,B 0,C 180,E1 16865.72,E2 16865.72} C_VEL
LIN {X 0,Y 370.28,Z 1201.781,A -85,B 0,C 180,E1 16861.594,E2 16861.594} C_VEL
LIN {X 0,Y 363.63,Z 1221.456,A -85,B 0,C 180,E1 16857.693,E2 16857.693} C_VEL
LIN {X 0,Y 359.271,Z 1236.662,A -85,B 0,C 180,E1 16854.151,E2 16854.151} C_VEL
LIN {X 0,Y 356.133,Z 1249.615,A -85,B 0,C 180,E1 16850.548,E2 16850.548} C_VEL
LIN {X 0,Y 354.178,Z 1259.361,A -85,B 0,C 180,E1 16847.245,E2 16847.245} C_VEL
LIN {X 0,Y 352.96,Z 1267.193,A -85,B 0,C 180,E1 16843.935,E2 16843.935} C_VEL
LIN {X 0,Y 352.356,Z 1273.167,A -85,B 0,C 180,E1 16840.631,E2 16840.631} C_VEL
LIN {X 0,Y 352.184,Z 1277.331,A -85,B 0,C 180,E1 16837.342,E2 16837.342} C_VEL
LIN {X 0,Y 352.235,Z 1279.625,A -85,B 0,C 180,E1 16834.235,E2 16834.235} C_VEL
LIN {X 0,Y 352.347,Z 1280.326,A -85,B 0,C 180,E1 16831.14,E2 16831.14} C_VEL
LIN {X 0,Y 352.384,Z 1279.448,A -85,B 0,C 180,E1 16828.051,E2 16828.051} C_VEL
LIN {X 0,Y 352.346,Z 1276.959,A -85,B 0,C 180,E1 16824.922,E2 16824.922} C_VEL
LIN {X 0,Y 352.339,Z 1272.719,A -85,B 0,C 180,E1 16821.681,E2 16821.681} C_VEL
LIN {X 0,Y 352.544,Z 1266.697,A -85,B 0,C 180,E1 16818.385,E2 16818.385} C_VEL
LIN {X 0,Y 353.147,Z 1258.858,A -85,B 0,C 180,E1 16815.072,E2 16815.072} C_VEL
LIN {X 0,Y 354.366,Z 1248.6,A -85,B 0,C 180,E1 16811.58,E2 16811.58} C_VEL
LIN {X 0,Y 356.21,Z 1236.808,A -85,B 0,C 180,E1 16808.255,E2 16808.255} C_VEL
LIN {X 0,Y 358.984,Z 1222.137,A -85,B 0,C 180,E1 16804.779,E2 16804.779} C_VEL
LIN {X 0,Y 362.509,Z 1205.759,A -85,B 0,C 180,E1 16801.502,E2 16801.502} C_VEL
LIN {X 0,Y 366.71,Z 1187.842,A -85,B 0,C 180,E1 16798.435,E2 16798.435} C_VEL
LIN {X 0,Y 371.834,Z 1167.311,A -85,B 0,C 180,E1 16795.434,E2 16795.434} C_VEL
LIN {X 0,Y 377.567,Z 1145.07,A -85,B 0,C 180,E1 16792.67,E2 16792.67} C_VEL
LIN {X 0,Y 384.222,Z 1119.532,A -85,B 0,C 180,E1 16790.003,E2 16790.003} C_VEL
LIN {X 0,Y 390.306,Z 1096.244,A -85,B 0,C 180,E1 16787.943,E2 16787.943} C_VEL
LIN {X 0,Y 396.869,Z 1070.769,A -85,B 0,C 180,E1 16786.047,E2 16786.047} C_VEL
LIN {X 0,Y 403.033,Z 1046.021,A -85,B 0,C 180,E1 16784.503,E2 16784.503} C_VEL
LIN {X 0,Y 409.078,Z 1020.075,A -85,B 0,C 180,E1 16783.199,E2 16783.199} C_VEL
LIN {X 0,Y 414.754,Z 992.319,A -85,B 0,C 180,E1 16782.057,E2 16782.057} C_VEL
LIN {X 0,Y 417.665,Z 975.288,A -85,B 0,C 180,E1 16781.469,E2 16781.469} C_VEL
LIN {X 0,Y 410.847,Z 954.975,A -85,B 0,C 180,E1 16779.772,E2 16779.772} C_VEL
LIN {X 0,Y 404.852,Z 932.686,A -85,B 0,C 180,E1 16778.107,E2 16778.107} C_VEL
LIN {X 0,Y 400.088,Z 908.548,A -85,B 0,C 180,E1 16776.462,E2 16776.462} C_VEL
LIN {X 0,Y 399.547,Z 904.545,A -85,B 0,C 180,E1 16776.2,E2 16776.2} C_VEL
LIN {X 0,Y 403.163,Z 878.968,A -85,B 0,C 180,E1 16773.189,E2 16773.189} C_VEL
LIN {X 0,Y 411.37,Z 840.996,A -85,B 0,C 180,E1 16768.957,E2 16768.957} C_VEL
LIN {X 0,Y 418.905,Z 807.81,A -85,B 0,C 180,E1 16765.231,E2 16765.231} C_VEL
LIN {X 0,Y 422.157,Z 792.892,A -85,B 0,C 180,E1 16763.529,E2 16763.529} C_VEL
LIN {X 0,Y 415.76,Z 775.535,A -85,B 0,C 180,E1 16759.969,E2 16759.969} C_VEL
LIN {X 0,Y 409.608,Z 759.722,A -85,B 0,C 180,E1 16756.449,E2 16756.449} C_VEL
LIN {X 0,Y 403.559,Z 744.998,A -85,B 0,C 180,E1 16752.885,E2 16752.885} C_VEL
LIN {X 0,Y 397.468,Z 730.715,A -85,B 0,C 180,E1 16749.119,E2 16749.119} C_VEL
LIN {X 0,Y 391.913,Z 718.311,A -85,B 0,C 180,E1 16745.564,E2 16745.564} C_VEL
LIN {X 0,Y 386.748,Z 707.066,A -85,B 0,C 180,E1 16742.074,E2 16742.074} C_VEL
LIN {X 0,Y 381.358,Z 695.535,A -85,B 0,C 180,E1 16738.197,E2 16738.197} C_VEL
LIN {X 0,Y 376.456,Z 685.682,A -85,B 0,C 180,E1 16734.513,E2 16734.513} C_VEL
LIN {X 0,Y 372.359,Z 677.296,A -85,B 0,C 180,E1 16731.164,E2 16731.164} C_VEL
LIN {X 0,Y 369.632,Z 672.131,A -85,B 0,C 180,E1 16728.927,E2 16728.927} C_VEL
LIN {X 0,Y 367.428,Z 667.721,A -85,B 0,C 180,E1 16726.946,E2 16726.946} C_VEL
LIN {X 0,Y 364.959,Z 662.944,A -85,B 0,C 180,E1 16724.651,E2 16724.651} C_VEL
LIN {X 0,Y 362.544,Z 658.274,A -85,B 0,C 180,E1 16722.339,E2 16722.339} C_VEL
LIN {X 0,Y 360.588,Z 654.604,A -85,B 0,C 180,E1 16720.395,E2 16720.395} C_VEL
LIN {X 0,Y 359.886,Z 653.292,A -85,B 0,C 180,E1 16719.678,E2 16719.678} C_VEL
LIN {X 0,Y 357.971,Z 649.816,A -85,B 0,C 180,E1 16717.674,E2 16717.674} C_VEL
LIN {X 0,Y 357.358,Z 648.461,A -85,B 0,C 180,E1 16716.938,E2 16716.938} C_VEL
LIN {X 0,Y 355.378,Z 645.272,A -85,B 0,C 180,E1 16714.858,E2 16714.858} C_VEL
LIN {X 0,Y 355.028,Z 643.751,A -85,B 0,C 180,E1 16714.117,E2 16714.117} C_VEL
LIN {X 0,Y 355.03,Z 643.745,A -85,B 0,C 180,E1 16710.099,E2 16710.099} C_VEL
LIN {X 0,Y 355.036,Z 643.739,A -85,B 0,C 180,E1 16705.888,E2 16705.888} C_VEL
LIN {X 0,Y 355.062,Z 643.942,A -85,B 0,C 180,E1 16705.67,E2 16705.67} C_VEL
LIN {X 0,Y 356.407,Z 647.33,A -85,B 0,C 180,E1 16704.999,E2 16704.999} C_VEL
LIN {X 0,Y 357.872,Z 649.434,A -85,B 0,C 180,E1 16704.468,E2 16704.468} C_VEL
LIN {X 0,Y 359.803,Z 653.008,A -85,B 0,C 180,E1 16703.693,E2 16703.693} C_VEL
LIN {X 0,Y 365.627,Z 663.999,A -85,B 0,C 180,E1 16701.426,E2 16701.426} C_VEL
LIN {X 0,Y 372.284,Z 677.592,A -85,B 0,C 180,E1 16698.85,E2 16698.85} C_VEL
LIN {X 0,Y 379.567,Z 694.853,A -85,B 0,C 180,E1 16695.936,E2 16695.936} C_VEL
LIN {X 0,Y 385.882,Z 712.44,A -85,B 0,C 180,E1 16693.271,E2 16693.271} C_VEL
LIN {X 0,Y 391.092,Z 730.068,A -85,B 0,C 180,E1 16690.852,E2 16690.852} C_VEL
LIN {X 0,Y 386.345,Z 778.034,A -85,B 0,C 180,E1 16686.713,E2 16686.713} C_VEL
LIN {X 0,Y 381.94,Z 825.838,A -85,B 0,C 180,E1 16682.632,E2 16682.632} C_VEL
LIN {X 0,Y 378.768,Z 867.779,A -85,B 0,C 180,E1 16679.197,E2 16679.197} C_VEL
LIN {X 0,Y 379.181,Z 874.758,A -85,B 0,C 180,E1 16679.009,E2 16679.009} C_VEL
LIN {X 0,Y 374.384,Z 1030.378,A -85,B 0,C 180,E1 16676.086,E2 16676.086} C_VEL
LIN {X 0,Y 373.913,Z 1048.559,A -85,B 0,C 180,E1 16675.568,E2 16675.568} C_VEL
LIN {X 0,Y 372.918,Z 1065.357,A -85,B 0,C 180,E1 16674.81,E2 16674.81} C_VEL
LIN {X 0,Y 371.474,Z 1081.436,A -85,B 0,C 180,E1 16673.81,E2 16673.81} C_VEL
LIN {X 0,Y 369.572,Z 1097.456,A -85,B 0,C 180,E1 16672.509,E2 16672.509} C_VEL
LIN {X 0,Y 367.4,Z 1112.242,A -85,B 0,C 180,E1 16670.968,E2 16670.968} C_VEL
LIN {X 0,Y 365.067,Z 1125.885,A -85,B 0,C 180,E1 16669.186,E2 16669.186} C_VEL
LIN {X 0,Y 362.691,Z 1138.422,A -85,B 0,C 180,E1 16667.154,E2 16667.154} C_VEL
LIN {X 0,Y 360.46,Z 1149.314,A -85,B 0,C 180,E1 16664.948,E2 16664.948} C_VEL
LIN {X 0,Y 358.464,Z 1158.662,A -85,B 0,C 180,E1 16662.564,E2 16662.564} C_VEL
LIN {X 0,Y 356.792,Z 1166.528,A -85,B 0,C 180,E1 16660.004,E2 16660.004} C_VEL
LIN {X 0,Y 355.568,Z 1172.511,A -85,B 0,C 180,E1 16657.43,E2 16657.43} C_VEL
LIN {X 0,Y 354.691,Z 1176.98,A -85,B 0,C 180,E1 16654.687,E2 16654.687} C_VEL
LIN {X 0,Y 354.185,Z 1179.83,A -85,B 0,C 180,E1 16651.777,E2 16651.777} C_VEL
LIN {X 0,Y 354.052,Z 1180.882,A -85,B 0,C 180,E1 16648.865,E2 16648.865} C_VEL
LIN {X 0,Y 354.233,Z 1180.209,A -85,B 0,C 180,E1 16646.113,E2 16646.113} C_VEL
LIN {X 0,Y 354.786,Z 1177.668,A -85,B 0,C 180,E1 16643.2,E2 16643.2} C_VEL
LIN {X 0,Y 355.794,Z 1173.235,A -85,B 0,C 180,E1 16640.29,E2 16640.29} C_VEL
LIN {X 0,Y 357.12,Z 1167.546,A -85,B 0,C 180,E1 16637.712,E2 16637.712} C_VEL
LIN {X 0,Y 358.903,Z 1159.933,A -85,B 0,C 180,E1 16635.147,E2 16635.147} C_VEL
LIN {X 0,Y 361.009,Z 1150.823,A -85,B 0,C 180,E1 16632.759,E2 16632.759} C_VEL
LIN {X 0,Y 363.366,Z 1140.254,A -85,B 0,C 180,E1 16630.549,E2 16630.549} C_VEL
LIN {X 0,Y 365.862,Z 1128.127,A -85,B 0,C 180,E1 16628.515,E2 16628.515} C_VEL
LIN {X 0,Y 368.301,Z 1114.855,A -85,B 0,C 180,E1 16626.731,E2 16626.731} C_VEL
LIN {X 0,Y 370.692,Z 1099.847,A -85,B 0,C 180,E1 16625.114,E2 16625.114} C_VEL
LIN {X 0,Y 372.684,Z 1084.729,A -85,B 0,C 180,E1 16623.828,E2 16623.828} C_VEL
LIN {X 0,Y 374.296,Z 1068.49,A -85,B 0,C 180,E1 16622.774,E2 16622.774} C_VEL
LIN {X 0,Y 375.474,Z 1050.725,A -85,B 0,C 180,E1 16621.935,E2 16621.935} C_VEL
LIN {X 0,Y 376.052,Z 1033.082,A -85,B 0,C 180,E1 16621.394,E2 16621.394} C_VEL
LIN {X 0,Y 378.077,Z 961.199,A -85,B 0,C 180,E1 16620.021,E2 16620.021} C_VEL
LIN {X 0,Y 380.97,Z 872.082,A -85,B 0,C 180,E1 16618.353,E2 16618.353} C_VEL
LIN {X 0,Y 380.655,Z 869.149,A -85,B 0,C 180,E1 16618.26,E2 16618.26} C_VEL
LIN {X 0,Y 381.012,Z 864.008,A -85,B 0,C 180,E1 16617.957,E2 16617.957} C_VEL
LIN {X 0,Y 380.466,Z 858.441,A -85,B 0,C 180,E1 16617.398,E2 16617.398} C_VEL
LIN {X 0,Y 376.153,Z 843.922,A -85,B 0,C 180,E1 16615.593,E2 16615.593} C_VEL
LIN {X 0,Y 376.006,Z 840.131,A -85,B 0,C 180,E1 16615.228,E2 16615.228} C_VEL
LIN {X 0,Y 378.808,Z 810.804,A -85,B 0,C 180,E1 16612.713,E2 16612.713} C_VEL
LIN {X 0,Y 380.541,Z 811.21,A -85,B 0,C 180,E1 16612.438,E2 16612.438} C_VEL
LIN {X 0,Y 383.514,Z 809.733,A -85,B 0,C 180,E1 16612.072,E2 16612.072} C_VEL
LIN {X 0,Y 387.617,Z 805.464,A -85,B 0,C 180,E1 16611.68,E2 16611.68} C_VEL
LIN {X 0,Y 388.636,Z 804.343,A -85,B 0,C 180,E1 16611.584,E2 16611.584} C_VEL
LIN {X 0,Y 392.801,Z 802.349,A -85,B 0,C 180,E1 16611.087,E2 16611.087} C_VEL
LIN {X 0,Y 397.554,Z 797.906,A -85,B 0,C 180,E1 16610.62,E2 16610.62} C_VEL
LIN {X 0,Y 398.626,Z 796.924,A -85,B 0,C 180,E1 16610.514,E2 16610.514} C_VEL
LIN {X 0,Y 403.678,Z 793.948,A -85,B 0,C 180,E1 16609.956,E2 16609.956} C_VEL
LIN {X 0,Y 409.026,Z 789.166,A -85,B 0,C 180,E1 16609.438,E2 16609.438} C_VEL
LIN {X 0,Y 414.994,Z 785.142,A -85,B 0,C 180,E1 16608.823,E2 16608.823} C_VEL
LIN {X 0,Y 418.727,Z 781.834,A -85,B 0,C 180,E1 16608.471,E2 16608.471} C_VEL
LIN {X 0,Y 398.619,Z 965.445,A -85,B 0,C 180,E1 16603.655,E2 16603.655} C_VEL
LIN {X 0,Y 395.393,Z 997.955,A -85,B 0,C 180,E1 16602.633,E2 16602.633} C_VEL
LIN {X 0,Y 392.4,Z 1021.352,A -85,B 0,C 180,E1 16601.64,E2 16601.64} C_VEL
LIN {X 0,Y 388.785,Z 1044.015,A -85,B 0,C 180,E1 16600.399,E2 16600.399} C_VEL
LIN {X 0,Y 384.768,Z 1065.269,A -85,B 0,C 180,E1 16598.968,E2 16598.968} C_VEL
LIN {X 0,Y 380.2,Z 1086.712,A -85,B 0,C 180,E1 16597.22,E2 16597.22} C_VEL
LIN {X 0,Y 375.542,Z 1106.496,A -85,B 0,C 180,E1 16595.294,E2 16595.294} C_VEL
LIN {X 0,Y 370.587,Z 1125.941,A -85,B 0,C 180,E1 16593.026,E2 16593.026} C_VEL
LIN {X 0,Y 365.92,Z 1143.233,A -85,B 0,C 180,E1 16590.639,E2 16590.639} C_VEL
LIN {X 0,Y 361.249,Z 1160.14,A -85,B 0,C 180,E1 16587.89,E2 16587.89} C_VEL
LIN {X 0,Y 357.105,Z 1175.157,A -85,B 0,C 180,E1 16585.012,E2 16585.012} C_VEL
LIN {X 0,Y 353.442,Z 1188.673,A -85,B 0,C 180,E1 16581.927,E2 16581.927} C_VEL
LIN {X 0,Y 350.34,Z 1200.803,A -85,B 0,C 180,E1 16578.635,E2 16578.635} C_VEL
LIN {X 0,Y 347.905,Z 1211.484,A -85,B 0,C 180,E1 16575.161,E2 16575.161} C_VEL
LIN {X 0,Y 346.2,Z 1220.311,A -85,B 0,C 180,E1 16571.664,E2 16571.664} C_VEL
LIN {X 0,Y 345.134,Z 1227.315,A -85,B 0,C 180,E1 16568.161,E2 16568.161} C_VEL
LIN {X 0,Y 344.548,Z 1233.014,A -85,B 0,C 180,E1 16564.494,E2 16564.494} C_VEL
LIN {X 0,Y 344.359,Z 1236.752,A -85,B 0,C 180,E1 16561.165,E2 16561.165} C_VEL
LIN {X 0,Y 344.342,Z 1239.364,A -85,B 0,C 180,E1 16557.504,E2 16557.504} C_VEL
LIN {X 0,Y 344.511,Z 1240.523,A -85,B 0,C 180,E1 16554.003,E2 16554.003} C_VEL
LIN {X 0,Y 344.92,Z 1240.183,A -85,B 0,C 180,E1 16550.32,E2 16550.32} C_VEL
LIN {X 0,Y 345.911,Z 1238.211,A -85,B 0,C 180,E1 16546.289,E2 16546.289} C_VEL
LIN {X 0,Y 347.649,Z 1234.718,A -85,B 0,C 180,E1 16542.422,E2 16542.422} C_VEL
LIN {X 0,Y 350.529,Z 1229.322,A -85,B 0,C 180,E1 16538.409,E2 16538.409} C_VEL
LIN {X 0,Y 354.649,Z 1222.045,A -85,B 0,C 180,E1 16534.446,E2 16534.446} C_VEL
LIN {X 0,Y 360.127,Z 1212.751,A -85,B 0,C 180,E1 16530.565,E2 16530.565} C_VEL
LIN {X 0,Y 366.716,Z 1201.809,A -85,B 0,C 180,E1 16526.953,E2 16526.953} C_VEL
LIN {X 0,Y 374.288,Z 1189.292,A -85,B 0,C 180,E1 16523.625,E2 16523.625} C_VEL
LIN {X 0,Y 382.661,Z 1175.255,A -85,B 0,C 180,E1 16520.583,E2 16520.583} C_VEL
LIN {X 0,Y 391.704,Z 1159.732,A -85,B 0,C 180,E1 16517.828,E2 16517.828} C_VEL
LIN {X 0,Y 401.866,Z 1142.008,A -85,B 0,C 180,E1 16515.24,E2 16515.24} C_VEL
LIN {X 0,Y 409.004,Z 1129.536,A -85,B 0,C 180,E1 16513.682,E2 16513.682} C_VEL
LIN {X 0,Y 395.992,Z 1146.385,A -85,B 0,C 180,E1 16511.614,E2 16511.614} C_VEL
LIN {X 0,Y 383.446,Z 1165.135,A -85,B 0,C 180,E1 16508.937,E2 16508.937} C_VEL
LIN {X 0,Y 371.32,Z 1187.258,A -85,B 0,C 180,E1 16505.321,E2 16505.321} C_VEL
LIN {X 0,Y 361.543,Z 1209.506,A -85,B 0,C 180,E1 16501.145,E2 16501.145} C_VEL
LIN {X 0,Y 355.214,Z 1227.019,A -85,B 0,C 180,E1 16497.314,E2 16497.314} C_VEL
LIN {X 0,Y 350.715,Z 1241.692,A -85,B 0,C 180,E1 16493.526,E2 16493.526} C_VEL
LIN {X 0,Y 347.7,Z 1253.396,A -85,B 0,C 180,E1 16489.887,E2 16489.887} C_VEL
LIN {X 0,Y 345.848,Z 1262.361,A -85,B 0,C 180,E1 16486.461,E2 16486.461} C_VEL
LIN {X 0,Y 344.734,Z 1269.584,A -85,B 0,C 180,E1 16482.951,E2 16482.951} C_VEL
LIN {X 0,Y 344.25,Z 1274.762,A -85,B 0,C 180,E1 16479.532,E2 16479.532} C_VEL
LIN {X 0,Y 344.197,Z 1278.073,A -85,B 0,C 180,E1 16476.173,E2 16476.173} C_VEL
LIN {X 0,Y 344.299,Z 1279.582,A -85,B 0,C 180,E1 16472.999,E2 16472.999} C_VEL
LIN {X 0,Y 344.405,Z 1279.51,A -85,B 0,C 180,E1 16469.836,E2 16469.836} C_VEL
LIN {X 0,Y 344.399,Z 1277.993,A -85,B 0,C 180,E1 16466.84,E2 16466.84} C_VEL
LIN {X 0,Y 344.353,Z 1274.84,A -85,B 0,C 180,E1 16463.667,E2 16463.667} C_VEL
LIN {X 0,Y 344.411,Z 1269.799,A -85,B 0,C 180,E1 16460.309,E2 16460.309} C_VEL
LIN {X 0,Y 344.766,Z 1262.995,A -85,B 0,C 180,E1 16456.928,E2 16456.928} C_VEL
LIN {X 0,Y 345.601,Z 1254.332,A -85,B 0,C 180,E1 16453.531,E2 16453.531} C_VEL
LIN {X 0,Y 347.213,Z 1242.787,A -85,B 0,C 180,E1 16449.852,E2 16449.852} C_VEL
LIN {X 0,Y 349.517,Z 1229.707,A -85,B 0,C 180,E1 16446.393,E2 16446.393} C_VEL
LIN {X 0,Y 352.63,Z 1214.672,A -85,B 0,C 180,E1 16443.023,E2 16443.023} C_VEL
LIN {X 0,Y 356.896,Z 1196.237,A -85,B 0,C 180,E1 16439.533,E2 16439.533} C_VEL
LIN {X 0,Y 361.984,Z 1175.884,A -85,B 0,C 180,E1 16436.278,E2 16436.278} C_VEL
LIN {X 0,Y 367.628,Z 1154.328,A -85,B 0,C 180,E1 16433.356,E2 16433.356} C_VEL
LIN {X 0,Y 373.47,Z 1132.297,A -85,B 0,C 180,E1 16430.817,E2 16430.817} C_VEL
LIN {X 0,Y 379.733,Z 1109.148,A -85,B 0,C 180,E1 16428.533,E2 16428.533} C_VEL
LIN {X 0,Y 386.434,Z 1083.872,A -85,B 0,C 180,E1 16426.427,E2 16426.427} C_VEL
LIN {X 0,Y 392.989,Z 1058.863,A -85,B 0,C 180,E1 16424.676,E2 16424.676} C_VEL
LIN {X 0,Y 399.288,Z 1033.531,A -85,B 0,C 180,E1 16423.225,E2 16423.225} C_VEL
LIN {X 0,Y 405.742,Z 1005.283,A -85,B 0,C 180,E1 16421.911,E2 16421.911} C_VEL
LIN {X 0,Y 410.954,Z 978.508,A -85,B 0,C 180,E1 16420.903,E2 16420.903} C_VEL
LIN {X 0,Y 410.643,Z 976.712,A -85,B 0,C 180,E1 16420.78,E2 16420.78} C_VEL
LIN {X 0,Y 403.376,Z 953.769,A -85,B 0,C 180,E1 16418.851,E2 16418.851} C_VEL
LIN {X 0,Y 397.665,Z 930.392,A -85,B 0,C 180,E1 16417.107,E2 16417.107} C_VEL
LIN {X 0,Y 393.321,Z 905.631,A -85,B 0,C 180,E1 16415.424,E2 16415.424} C_VEL
LIN {X 0,Y 392.987,Z 902.226,A -85,B 0,C 180,E1 16415.19,E2 16415.19} C_VEL
LIN {X 0,Y 397.309,Z 876.15,A -85,B 0,C 180,E1 16412.12,E2 16412.12} C_VEL
LIN {X 0,Y 405.296,Z 840.466,A -85,B 0,C 180,E1 16408.113,E2 16408.113} C_VEL
LIN {X 0,Y 412.887,Z 807.878,A -85,B 0,C 180,E1 16404.424,E2 16404.424} C_VEL
LIN {X 0,Y 415.459,Z 796.446,A -85,B 0,C 180,E1 16403.097,E2 16403.097} C_VEL
LIN {X 0,Y 408.994,Z 778.832,A -85,B 0,C 180,E1 16399.42,E2 16399.42} C_VEL
LIN {X 0,Y 402.665,Z 762.477,A -85,B 0,C 180,E1 16395.704,E2 16395.704} C_VEL
LIN {X 0,Y 396.166,Z 746.705,A -85,B 0,C 180,E1 16391.797,E2 16391.797} C_VEL
LIN {X 0,Y 390.324,Z 733.013,A -85,B 0,C 180,E1 16388.1,E2 16388.1} C_VEL
LIN {X 0,Y 384.594,Z 720.255,A -85,B 0,C 180,E1 16384.324,E2 16384.324} C_VEL
LIN {X 0,Y 379.298,Z 708.729,A -85,B 0,C 180,E1 16380.604,E2 16380.604} C_VEL
LIN {X 0,Y 373.787,Z 696.944,A -85,B 0,C 180,E1 16376.473,E2 16376.473} C_VEL
LIN {X 0,Y 368.922,Z 687.198,A -85,B 0,C 180,E1 16372.681,E2 16372.681} C_VEL
LIN {X 0,Y 366.38,Z 682.213,A -85,B 0,C 180,E1 16370.576,E2 16370.576} C_VEL
LIN {X 0,Y 364.068,Z 677.649,A -85,B 0,C 180,E1 16368.595,E2 16368.595} C_VEL
LIN {X 0,Y 361.816,Z 673.213,A -85,B 0,C 180,E1 16366.577,E2 16366.577} C_VEL
LIN {X 0,Y 359.694,Z 668.917,A -85,B 0,C 180,E1 16364.522,E2 16364.522} C_VEL
LIN {X 0,Y 357.212,Z 664.159,A -85,B 0,C 180,E1 16362.112,E2 16362.112} C_VEL
LIN {X 0,Y 355.255,Z 660.195,A -85,B 0,C 180,E1 16360.054,E2 16360.054} C_VEL
LIN {X 0,Y 352.781,Z 655.831,A -85,B 0,C 180,E1 16357.503,E2 16357.503} C_VEL
LIN {X 0,Y 352.154,Z 654.496,A -85,B 0,C 180,E1 16356.754,E2 16356.754} C_VEL
LIN {X 0,Y 350.202,Z 651.224,A -85,B 0,C 180,E1 16354.642,E2 16354.642} C_VEL
LIN {X 0,Y 349.723,Z 649.735,A -85,B 0,C 180,E1 16353.858,E2 16353.858} C_VEL
LIN {X 0,Y 347.531,Z 646.513,A -85,B 0,C 180,E1 16351.471,E2 16351.471} C_VEL
LIN {X 0,Y 347.094,Z 644.739,A -85,B 0,C 180,E1 16350.451,E2 16350.451} C_VEL
LIN {X 0,Y 347.107,Z 644.851,A -85,B 0,C 180,E1 16347.256,E2 16347.256} C_VEL
LIN {X 0,Y 348.405,Z 648.233,A -85,B 0,C 180,E1 16346.563,E2 16346.563} C_VEL
LIN {X 0,Y 350.058,Z 650.344,A -85,B 0,C 180,E1 16345.955,E2 16345.955} C_VEL
LIN {X 0,Y 351.844,Z 653.864,A -85,B 0,C 180,E1 16345.165,E2 16345.165} C_VEL
LIN {X 0,Y 357.692,Z 664.435,A -85,B 0,C 180,E1 16342.81,E2 16342.81} C_VEL
LIN {X 0,Y 365.019,Z 679.295,A -85,B 0,C 180,E1 16339.837,E2 16339.837} C_VEL
LIN {X 0,Y 372.108,Z 695.702,A -85,B 0,C 180,E1 16336.957,E2 16336.957} C_VEL
LIN {X 0,Y 378.176,Z 712.234,A -85,B 0,C 180,E1 16334.34,E2 16334.34} C_VEL
LIN {X 0,Y 383.801,Z 730.56,A -85,B 0,C 180,E1 16331.72,E2 16331.72} C_VEL
LIN {X 0,Y 384.434,Z 733.56,A -85,B 0,C 180,E1 16331.345,E2 16331.345} C_VEL
LIN {X 0,Y 379.624,Z 780.17,A -85,B 0,C 180,E1 16327.283,E2 16327.283} C_VEL
LIN {X 0,Y 375.024,Z 828.473,A -85,B 0,C 180,E1 16323.129,E2 16323.129} C_VEL
LIN {X 0,Y 371.86,Z 868.639,A -85,B 0,C 180,E1 16319.807,E2 16319.807} C_VEL
LIN {X 0,Y 372.262,Z 875.637,A -85,B 0,C 180,E1 16319.615,E2 16319.615} C_VEL
LIN {X 0,Y 367.289,Z 1030.788,A -85,B 0,C 180,E1 16316.653,E2 16316.653} C_VEL
LIN {X 0,Y 366.803,Z 1049.16,A -85,B 0,C 180,E1 16316.127,E2 16316.127} C_VEL
LIN {X 0,Y 365.797,Z 1065.731,A -85,B 0,C 180,E1 16315.374,E2 16315.374} C_VEL
LIN {X 0,Y 364.233,Z 1082.544,A -85,B 0,C 180,E1 16314.314,E2 16314.314} C_VEL
LIN {X 0,Y 362.256,Z 1098.561,A -85,B 0,C 180,E1 16312.987,E2 16312.987} C_VEL
LIN {X 0,Y 360.005,Z 1113.29,A -85,B 0,C 180,E1 16311.419,E2 16311.419} C_VEL
LIN {X 0,Y 357.584,Z 1126.918,A -85,B 0,C 180,E1 16309.603,E2 16309.603} C_VEL
LIN {X 0,Y 355.117,Z 1139.443,A -85,B 0,C 180,E1 16307.532,E2 16307.532} C_VEL
LIN {X 0,Y 352.796,Z 1150.319,A -85,B 0,C 180,E1 16305.28,E2 16305.28} C_VEL
LIN {X 0,Y 350.688,Z 1159.793,A -85,B 0,C 180,E1 16302.807,E2 16302.807} C_VEL
LIN {X 0,Y 348.973,Z 1167.517,A -85,B 0,C 180,E1 16300.23,E2 16300.23} C_VEL
LIN {X 0,Y 347.694,Z 1173.491,A -85,B 0,C 180,E1 16297.599,E2 16297.599} C_VEL
LIN {X 0,Y 346.776,Z 1177.949,A -85,B 0,C 180,E1 16294.794,E2 16294.794} C_VEL
LIN {X 0,Y 346.248,Z 1180.792,A -85,B 0,C 180,E1 16291.818,E2 16291.818} C_VEL
LIN {X 0,Y 346.109,Z 1181.837,A -85,B 0,C 180,E1 16288.839,E2 16288.839} C_VEL
LIN {X 0,Y 346.302,Z 1181.153,A -85,B 0,C 180,E1 16286.024,E2 16286.024} C_VEL
LIN {X 0,Y 346.887,Z 1178.605,A -85,B 0,C 180,E1 16283.044,E2 16283.044} C_VEL
LIN {X 0,Y 347.949,Z 1174.164,A -85,B 0,C 180,E1 16280.069,E2 16280.069} C_VEL
LIN {X 0,Y 349.354,Z 1168.425,A -85,B 0,C 180,E1 16277.418,E2 16277.418} C_VEL
LIN {X 0,Y 351.21,Z 1160.84,A -85,B 0,C 180,E1 16274.814,E2 16274.814} C_VEL
LIN {X 0,Y 353.412,Z 1151.719,A -85,B 0,C 180,E1 16272.376,E2 16272.376} C_VEL
LIN {X 0,Y 355.868,Z 1141.136,A -85,B 0,C 180,E1 16270.123,E2 16270.123} C_VEL
LIN {X 0,Y 358.465,Z 1128.986,A -85,B 0,C 180,E1 16268.049,E2 16268.049} C_VEL
LIN {X 0,Y 360.979,Z 1115.818,A -85,B 0,C 180,E1 16266.247,E2 16266.247} C_VEL
LIN {X 0,Y 363.348,Z 1101.542,A -85,B 0,C 180,E1 16264.674,E2 16264.674} C_VEL
LIN {X 0,Y 365.456,Z 1086.262,A -85,B 0,C 180,E1 16263.337,E2 16263.337} C_VEL
LIN {X 0,Y 367.166,Z 1069.889,A -85,B 0,C 180,E1 16262.244,E2 16262.244} C_VEL
LIN {X 0,Y 368.39,Z 1052.413,A -85,B 0,C 180,E1 16261.396,E2 16261.396} C_VEL
LIN {X 0,Y 369.023,Z 1034.815,A -85,B 0,C 180,E1 16260.835,E2 16260.835} C_VEL
LIN {X 0,Y 370.73,Z 974.091,A -85,B 0,C 180,E1 16259.645,E2 16259.645} C_VEL
LIN {X 0,Y 374.15,Z 872.934,A -85,B 0,C 180,E1 16257.722,E2 16257.722} C_VEL
LIN {X 0,Y 373.669,Z 868.082,A -85,B 0,C 180,E1 16257.552,E2 16257.552} C_VEL
LIN {X 0,Y 376.006,Z 840.131,A -85,B 0,C 180,E1 16255.228,E2 16255.228} C_VEL
LIN {X 0,Y 375.738,Z 836.309,A -85,B 0,C 180,E1 16254.795,E2 16254.795} C_VEL
LIN {X 0,Y 373.742,Z 829.807,A -85,B 0,C 180,E1 16253.595,E2 16253.595} C_VEL
LIN {X 0,Y 373.936,Z 826.676,A -85,B 0,C 180,E1 16252.948,E2 16252.948} C_VEL
LIN {X 0,Y 375.597,Z 824.285,A -85,B 0,C 180,E1 16252.536,E2 16252.536} C_VEL
LIN {X 0,Y 375.835,Z 824.083,A -85,B 0,C 180,E1 16252.508,E2 16252.508} C_VEL
LIN {X 0,Y 379.777,Z 819.868,A -85,B 0,C 180,E1 16252.137,E2 16252.137} C_VEL
LIN {X 0,Y 380.617,Z 818.824,A -85,B 0,C 180,E1 16252.066,E2 16252.066} C_VEL
LIN {X 0,Y 384.569,Z 817.036,A -85,B 0,C 180,E1 16251.579,E2 16251.579} C_VEL
LIN {X 0,Y 389.245,Z 812.906,A -85,B 0,C 180,E1 16251.11,E2 16251.11} C_VEL
LIN {X 0,Y 391.099,Z 811.137,A -85,B 0,C 180,E1 16250.933,E2 16250.933} C_VEL
LIN {X 0,Y 396.213,Z 807.944,A -85,B 0,C 180,E1 16250.367,E2 16250.367} C_VEL
LIN {X 0,Y 400.786,Z 803.706,A -85,B 0,C 180,E1 16249.933,E2 16249.933} C_VEL
LIN {X 0,Y 406.756,Z 799.82,A -85,B 0,C 180,E1 16249.303,E2 16249.303} C_VEL
LIN {X 0,Y 411.228,Z 795.867,A -85,B 0,C 180,E1 16248.881,E2 16248.881} C_VEL
LIN {X 0,Y 391.33,Z 972.101,A -85,B 0,C 180,E1 16244.113,E2 16244.113} C_VEL
LIN {X 0,Y 388.17,Z 1002.205,A -85,B 0,C 180,E1 16243.104,E2 16243.104} C_VEL
LIN {X 0,Y 385.025,Z 1025.237,A -85,B 0,C 180,E1 16242.068,E2 16242.068} C_VEL
LIN {X 0,Y 381.443,Z 1046.785,A -85,B 0,C 180,E1 16240.846,E2 16240.846} C_VEL
LIN {X 0,Y 377.139,Z 1068.555,A -85,B 0,C 180,E1 16239.32,E2 16239.32} C_VEL
LIN {X 0,Y 372.488,Z 1089.509,A -85,B 0,C 180,E1 16237.543,E2 16237.543} C_VEL
LIN {X 0,Y 367.525,Z 1109.813,A -85,B 0,C 180,E1 16235.481,E2 16235.481} C_VEL
LIN {X 0,Y 362.559,Z 1128.778,A -85,B 0,C 180,E1 16233.192,E2 16233.192} C_VEL
LIN {X 0,Y 357.55,Z 1146.795,A -85,B 0,C 180,E1 16230.595,E2 16230.595} C_VEL
LIN {X 0,Y 352.995,Z 1162.808,A -85,B 0,C 180,E1 16227.864,E2 16227.864} C_VEL
LIN {X 0,Y 348.617,Z 1178.242,A -85,B 0,C 180,E1 16224.756,E2 16224.756} C_VEL
LIN {X 0,Y 344.995,Z 1191.49,A -85,B 0,C 180,E1 16221.597,E2 16221.597} C_VEL
LIN {X 0,Y 341.966,Z 1203.25,A -85,B 0,C 180,E1 16218.232,E2 16218.232} C_VEL
LIN {X 0,Y 339.585,Z 1213.593,A -85,B 0,C 180,E1 16214.668,E2 16214.668} C_VEL
LIN {X 0,Y 337.974,Z 1222.126,A -85,B 0,C 180,E1 16211.087,E2 16211.087} C_VEL
LIN {X 0,Y 336.991,Z 1228.925,A -85,B 0,C 180,E1 16207.502,E2 16207.502} C_VEL
LIN {X 0,Y 336.505,Z 1234.108,A -85,B 0,C 180,E1 16203.919,E2 16203.919} C_VEL
LIN {X 0,Y 336.359,Z 1237.9,A -85,B 0,C 180,E1 16200.341,E2 16200.341} C_VEL
LIN {X 0,Y 336.376,Z 1240.155,A -85,B 0,C 180,E1 16196.762,E2 16196.762} C_VEL
LIN {X 0,Y 336.601,Z 1241.15,A -85,B 0,C 180,E1 16193.004,E2 16193.004} C_VEL
LIN {X 0,Y 337.162,Z 1240.683,A -85,B 0,C 180,E1 16189.232,E2 16189.232} C_VEL
LIN {X 0,Y 338.336,Z 1238.594,A -85,B 0,C 180,E1 16185.276,E2 16185.276} C_VEL
LIN {X 0,Y 340.494,Z 1234.762,A -85,B 0,C 180,E1 16181.154,E2 16181.154} C_VEL
LIN {X 0,Y 343.845,Z 1229.167,A -85,B 0,C 180,E1 16177.066,E2 16177.066} C_VEL
LIN {X 0,Y 348.308,Z 1222.095,A -85,B 0,C 180,E1 16173.211,E2 16173.211} C_VEL
LIN {X 0,Y 354.098,Z 1213.214,A -85,B 0,C 180,E1 16169.451,E2 16169.451} C_VEL
LIN {X 0,Y 361.237,Z 1202.37,A -85,B 0,C 180,E1 16165.813,E2 16165.813} C_VEL
LIN {X 0,Y 369.371,Z 1190.001,A -85,B 0,C 180,E1 16162.477,E2 16162.477} C_VEL
LIN {X 0,Y 378.323,Z 1176.204,A -85,B 0,C 180,E1 16159.446,E2 16159.446} C_VEL
LIN {X 0,Y 388.491,Z 1160.294,A -85,B 0,C 180,E1 16156.591,E2 16156.591} C_VEL
LIN {X 0,Y 399.97,Z 1142.312,A -85,B 0,C 180,E1 16153.947,E2 16153.947} C_VEL
LIN {X 0,Y 400.857,Z 1140.894,A -85,B 0,C 180,E1 16153.756,E2 16153.756} C_VEL
LIN {X 0,Y 387.19,Z 1157.492,A -85,B 0,C 180,E1 16151.504,E2 16151.504} C_VEL
LIN {X 0,Y 374.45,Z 1175.409,A -85,B 0,C 180,E1 16148.673,E2 16148.673} C_VEL
LIN {X 0,Y 361.784,Z 1197.347,A -85,B 0,C 180,E1 16144.706,E2 16144.706} C_VEL
LIN {X 0,Y 351.896,Z 1218.794,A -85,B 0,C 180,E1 16140.196,E2 16140.196} C_VEL
LIN {X 0,Y 345.671,Z 1235.357,A -85,B 0,C 180,E1 16136.085,E2 16136.085} C_VEL
LIN {X 0,Y 341.531,Z 1248.474,A -85,B 0,C 180,E1 16132.192,E2 16132.192} C_VEL
LIN {X 0,Y 338.918,Z 1258.444,A -85,B 0,C 180,E1 16128.582,E2 16128.582} C_VEL
LIN {X 0,Y 337.274,Z 1266.436,A -85,B 0,C 180,E1 16124.949,E2 16124.949} C_VEL
LIN {X 0,Y 336.46,Z 1272.233,A -85,B 0,C 180,E1 16121.487,E2 16121.487} C_VEL
LIN {X 0,Y 336.189,Z 1276.263,A -85,B 0,C 180,E1 16118.038,E2 16118.038} C_VEL
LIN {X 0,Y 336.244,Z 1278.49,A -85,B 0,C 180,E1 16114.778,E2 16114.778} C_VEL
LIN {X 0,Y 336.378,Z 1279.137,A -85,B 0,C 180,E1 16111.535,E2 16111.535} C_VEL
LIN {X 0,Y 336.439,Z 1278.299,A -85,B 0,C 180,E1 16108.47,E2 16108.47} C_VEL
LIN {X 0,Y 336.41,Z 1275.859,A -85,B 0,C 180,E1 16105.229,E2 16105.229} C_VEL
LIN {X 0,Y 336.385,Z 1271.82,A -85,B 0,C 180,E1 16101.972,E2 16101.972} C_VEL
LIN {X 0,Y 336.569,Z 1265.839,A -85,B 0,C 180,E1 16098.521,E2 16098.521} C_VEL
LIN {X 0,Y 337.168,Z 1258.043,A -85,B 0,C 180,E1 16095.051,E2 16095.051} C_VEL
LIN {X 0,Y 338.424,Z 1247.768,A -85,B 0,C 180,E1 16091.395,E2 16091.395} C_VEL
LIN {X 0,Y 340.351,Z 1235.986,A -85,B 0,C 180,E1 16087.914,E2 16087.914} C_VEL
LIN {X 0,Y 343.268,Z 1221.275,A -85,B 0,C 180,E1 16084.28,E2 16084.28} C_VEL
LIN {X 0,Y 346.777,Z 1205.767,A -85,B 0,C 180,E1 16081.029,E2 16081.029} C_VEL
LIN {X 0,Y 351.388,Z 1187.094,A -85,B 0,C 180,E1 16077.686,E2 16077.686} C_VEL
LIN {X 0,Y 356.97,Z 1165.853,A -85,B 0,C 180,E1 16074.467,E2 16074.467} C_VEL
LIN {X 0,Y 363.379,Z 1142.309,A -85,B 0,C 180,E1 16071.462,E2 16071.462} C_VEL
LIN {X 0,Y 370.454,Z 1116.483,A -85,B 0,C 180,E1 16068.709,E2 16068.709} C_VEL
LIN {X 0,Y 377.126,Z 1092.276,A -85,B 0,C 180,E1 16066.53,E2 16066.53} C_VEL
LIN {X 0,Y 384.039,Z 1066.596,A -85,B 0,C 180,E1 16064.599,E2 16064.599} C_VEL
LIN {X 0,Y 390.811,Z 1040.575,A -85,B 0,C 180,E1 16062.972,E2 16062.972} C_VEL
LIN {X 0,Y 397.023,Z 1015.099,A -85,B 0,C 180,E1 16061.685,E2 16061.685} C_VEL
LIN {X 0,Y 402.854,Z 987.238,A -85,B 0,C 180,E1 16060.529,E2 16060.529} C_VEL
LIN {X 0,Y 404.227,Z 979.907,A -85,B 0,C 180,E1 16060.258,E2 16060.258} C_VEL
LIN {X 0,Y 397.133,Z 956.513,A -85,B 0,C 180,E1 16058.229,E2 16058.229} C_VEL
LIN {X 0,Y 391.307,Z 931.725,A -85,B 0,C 180,E1 16056.346,E2 16056.346} C_VEL
LIN {X 0,Y 387.146,Z 906.351,A -85,B 0,C 180,E1 16054.614,E2 16054.614} C_VEL
LIN {X 0,Y 386.509,Z 900.127,A -85,B 0,C 180,E1 16054.196,E2 16054.196} C_VEL
LIN {X 0,Y 391.889,Z 871.612,A -85,B 0,C 180,E1 16050.854,E2 16050.854} C_VEL
LIN {X 0,Y 400.023,Z 836.864,A -85,B 0,C 180,E1 16046.9,E2 16046.9} C_VEL
LIN {X 0,Y 408.051,Z 803.543,A -85,B 0,C 180,E1 16043.083,E2 16043.083} C_VEL
LIN {X 0,Y 408.781,Z 800.055,A -85,B 0,C 180,E1 16042.659,E2 16042.659} C_VEL
LIN {X 0,Y 402.46,Z 782.723,A -85,B 0,C 180,E1 16038.994,E2 16038.994} C_VEL
LIN {X 0,Y 396.357,Z 766.901,A -85,B 0,C 180,E1 16035.36,E2 16035.36} C_VEL
LIN {X 0,Y 390.122,Z 751.643,A -85,B 0,C 180,E1 16031.532,E2 16031.532} C_VEL
LIN {X 0,Y 384.526,Z 738.399,A -85,B 0,C 180,E1 16027.922,E2 16027.922} C_VEL
LIN {X 0,Y 378.828,Z 725.58,A -85,B 0,C 180,E1 16024.087,E2 16024.087} C_VEL
LIN {X 0,Y 373.758,Z 714.424,A -85,B 0,C 180,E1 16020.46,E2 16020.46} C_VEL
LIN {X 0,Y 368.59,Z 703.501,A -85,B 0,C 180,E1 16016.599,E2 16016.599} C_VEL
LIN {X 0,Y 363.836,Z 693.538,A -85,B 0,C 180,E1 16012.768,E2 16012.768} C_VEL
LIN {X 0,Y 360.782,Z 687.683,A -85,B 0,C 180,E1 16010.267,E2 16010.267} C_VEL
LIN {X 0,Y 358.716,Z 683.498,A -85,B 0,C 180,E1 16008.422,E2 16008.422} C_VEL
LIN {X 0,Y 356.445,Z 679.024,A -85,B 0,C 180,E1 16006.371,E2 16006.371} C_VEL
LIN {X 0,Y 354.244,Z 674.637,A -85,B 0,C 180,E1 16004.25,E2 16004.25} C_VEL
LIN {X 0,Y 351.982,Z 670.156,A -85,B 0,C 180,E1 16001.962,E2 16001.962} C_VEL
LIN {X 0,Y 349.435,Z 665.299,A -85,B 0,C 180,E1 15999.332,E2 15999.332} C_VEL
LIN {X 0,Y 347.429,Z 661.258,A -85,B 0,C 180,E1 15997.058,E2 15997.058} C_VEL
LIN {X 0,Y 344.98,Z 657.01,A -85,B 0,C 180,E1 15994.336,E2 15994.336} C_VEL
LIN {X 0,Y 344.294,Z 655.558,A -85,B 0,C 180,E1 15993.433,E2 15993.433} C_VEL
LIN {X 0,Y 342.205,Z 651.875,A -85,B 0,C 180,E1 15990.879,E2 15990.879} C_VEL
LIN {X 0,Y 341.576,Z 650.53,A -85,B 0,C 180,E1 15989.962,E2 15989.962} C_VEL
LIN {X 0,Y 340.181,Z 648.749,A -85,B 0,C 180,E1 15988.354,E2 15988.354} C_VEL
LIN {X 0,Y 342.166,Z 651.28,A -85,B 0,C 180,E1 15987.572,E2 15987.572} C_VEL
LIN {X 0,Y 344.055,Z 654.993,A -85,B 0,C 180,E1 15986.683,E2 15986.683} C_VEL
LIN {X 0,Y 345.212,Z 656.773,A -85,B 0,C 180,E1 15986.212,E2 15986.212} C_VEL
LIN {X 0,Y 350.394,Z 666.298,A -85,B 0,C 180,E1 15983.996,E2 15983.996} C_VEL
LIN {X 0,Y 356.812,Z 678.931,A -85,B 0,C 180,E1 15981.324,E2 15981.324} C_VEL
LIN {X 0,Y 363.876,Z 694.661,A -85,B 0,C 180,E1 15978.364,E2 15978.364} C_VEL
LIN {X 0,Y 370.198,Z 711.145,A -85,B 0,C 180,E1 15975.609,E2 15975.609} C_VEL
LIN {X 0,Y 375.643,Z 728.086,A -85,B 0,C 180,E1 15973.057,E2 15973.057} C_VEL
LIN {X 0,Y 377.872,Z 736.279,A -85,B 0,C 180,E1 15971.92,E2 15971.92} C_VEL
LIN {X 0,Y 373.05,Z 781.368,A -85,B 0,C 180,E1 15967.958,E2 15967.958} C_VEL
LIN {X 0,Y 368.246,Z 830.226,A -85,B 0,C 180,E1 15963.726,E2 15963.726} C_VEL
LIN {X 0,Y 365.016,Z 869.692,A -85,B 0,C 180,E1 15960.435,E2 15960.435} C_VEL
LIN {X 0,Y 365.389,Z 876.513,A -85,B 0,C 180,E1 15960.244,E2 15960.244} C_VEL
LIN {X 0,Y 360.231,Z 1031.044,A -85,B 0,C 180,E1 15957.246,E2 15957.246} C_VEL
LIN {X 0,Y 359.733,Z 1049.593,A -85,B 0,C 180,E1 15956.714,E2 15956.714} C_VEL
LIN {X 0,Y 358.697,Z 1066.289,A -85,B 0,C 180,E1 15955.951,E2 15955.951} C_VEL
LIN {X 0,Y 357.142,Z 1082.573,A -85,B 0,C 180,E1 15954.917,E2 15954.917} C_VEL
LIN {X 0,Y 355.158,Z 1098.254,A -85,B 0,C 180,E1 15953.614,E2 15953.614} C_VEL
LIN {X 0,Y 352.867,Z 1113.047,A -85,B 0,C 180,E1 15952.05,E2 15952.05} C_VEL
LIN {X 0,Y 350.333,Z 1126.878,A -85,B 0,C 180,E1 15950.2,E2 15950.2} C_VEL
LIN {X 0,Y 347.743,Z 1139.569,A -85,B 0,C 180,E1 15948.089,E2 15948.089} C_VEL
LIN {X 0,Y 345.308,Z 1150.645,A -85,B 0,C 180,E1 15945.792,E2 15945.792} C_VEL
LIN {X 0,Y 343.113,Z 1160.102,A -85,B 0,C 180,E1 15943.307,E2 15943.307} C_VEL
LIN {X 0,Y 341.259,Z 1168.063,A -85,B 0,C 180,E1 15940.635,E2 15940.635} C_VEL
LIN {X 0,Y 339.823,Z 1174.471,A -85,B 0,C 180,E1 15937.776,E2 15937.776} C_VEL
LIN {X 0,Y 338.862,Z 1178.917,A -85,B 0,C 180,E1 15934.906,E2 15934.906} C_VEL
LIN {X 0,Y 338.31,Z 1181.753,A -85,B 0,C 180,E1 15931.861,E2 15931.861} C_VEL
LIN {X 0,Y 338.167,Z 1182.792,A -85,B 0,C 180,E1 15928.812,E2 15928.812} C_VEL
LIN {X 0,Y 338.372,Z 1182.098,A -85,B 0,C 180,E1 15925.931,E2 15925.931} C_VEL
LIN {X 0,Y 338.991,Z 1179.542,A -85,B 0,C 180,E1 15922.882,E2 15922.882} C_VEL
LIN {X 0,Y 340.11,Z 1175.094,A -85,B 0,C 180,E1 15919.838,E2 15919.838} C_VEL
LIN {X 0,Y 341.619,Z 1169.217,A -85,B 0,C 180,E1 15917.076,E2 15917.076} C_VEL
LIN {X 0,Y 343.547,Z 1161.681,A -85,B 0,C 180,E1 15914.446,E2 15914.446} C_VEL
LIN {X 0,Y 346.003,Z 1151.937,A -85,B 0,C 180,E1 15911.812,E2 15911.812} C_VEL
LIN {X 0,Y 348.592,Z 1141.193,A -85,B 0,C 180,E1 15909.514,E2 15909.514} C_VEL
LIN {X 0,Y 351.313,Z 1128.769,A -85,B 0,C 180,E1 15907.402,E2 15907.402} C_VEL
LIN {X 0,Y 354.094,Z 1114.591,A -85,B 0,C 180,E1 15905.472,E2 15905.472} C_VEL
LIN {X 0,Y 356.567,Z 1099.87,A -85,B 0,C 180,E1 15903.877,E2 15903.877} C_VEL
LIN {X 0,Y 358.61,Z 1084.913,A -85,B 0,C 180,E1 15902.607,E2 15902.607} C_VEL
LIN {X 0,Y 360.319,Z 1068.458,A -85,B 0,C 180,E1 15901.534,E2 15901.534} C_VEL
LIN {X 0,Y 361.516,Z 1051.154,A -85,B 0,C 180,E1 15900.715,E2 15900.715} C_VEL
LIN {X 0,Y 362.086,Z 1033.422,A -85,B 0,C 180,E1 15900.179,E2 15900.179} C_VEL
LIN {X 0,Y 364.508,Z 956.01,A -85,B 0,C 180,E1 15898.658,E2 15898.658} C_VEL
LIN {X 0,Y 367.391,Z 873.929,A -85,B 0,C 180,E1 15897.073,E2 15897.073} C_VEL
LIN {X 0,Y 366.929,Z 868.844,A -85,B 0,C 180,E1 15896.88,E2 15896.88} C_VEL
LIN {X 0,Y 370.911,Z 825.279,A -85,B 0,C 180,E1 15893.184,E2 15893.184} C_VEL
LIN {X 0,Y 372.807,Z 825.689,A -85,B 0,C 180,E1 15892.88,E2 15892.88} C_VEL
LIN {X 0,Y 375.835,Z 824.083,A -85,B 0,C 180,E1 15892.508,E2 15892.508} C_VEL
LIN {X 0,Y 380.116,Z 821.663,A -85,B 0,C 180,E1 15892.003,E2 15892.003} C_VEL
LIN {X 0,Y 392.483,Z 818.234,A -85,B 0,C 180,E1 15890.428,E2 15890.428} C_VEL
LIN {X 0,Y 393.598,Z 817.697,A -85,B 0,C 180,E1 15890.3,E2 15890.3} C_VEL
LIN {X 0,Y 399.494,Z 813.61,A -85,B 0,C 180,E1 15889.683,E2 15889.683} C_VEL
LIN {X 0,Y 403.55,Z 810.109,A -85,B 0,C 180,E1 15889.3,E2 15889.3} C_VEL
LIN {X 0,Y 383.701,Z 982.071,A -85,B 0,C 180,E1 15884.468,E2 15884.468} C_VEL
LIN {X 0,Y 380.95,Z 1006.279,A -85,B 0,C 180,E1 15883.586,E2 15883.586} C_VEL
LIN {X 0,Y 377.445,Z 1030.139,A -85,B 0,C 180,E1 15882.444,E2 15882.444} C_VEL
LIN {X 0,Y 373.245,Z 1053.545,A -85,B 0,C 180,E1 15881.021,E2 15881.021} C_VEL
LIN {X 0,Y 368.67,Z 1075.478,A -85,B 0,C 180,E1 15879.377,E2 15879.377} C_VEL
LIN {X 0,Y 363.843,Z 1096.186,A -85,B 0,C 180,E1 15877.497,E2 15877.497} C_VEL
LIN {X 0,Y 358.744,Z 1115.978,A -85,B 0,C 180,E1 15875.334,E2 15875.334} C_VEL
LIN {X 0,Y 353.707,Z 1134.246,A -85,B 0,C 180,E1 15872.969,E2 15872.969} C_VEL
LIN {X 0,Y 348.745,Z 1151.647,A -85,B 0,C 180,E1 15870.306,E2 15870.306} C_VEL
LIN {X 0,Y 344.231,Z 1167.171,A -85,B 0,C 180,E1 15867.507,E2 15867.507} C_VEL
LIN {X 0,Y 340.132,Z 1181.273,A -85,B 0,C 180,E1 15864.488,E2 15864.488} C_VEL
LIN {X 0,Y 336.374,Z 1194.728,A -85,B 0,C 180,E1 15861.081,E2 15861.081} C_VEL
LIN {X 0,Y 333.451,Z 1206.15,A -85,B 0,C 180,E1 15857.63,E2 15857.63} C_VEL
LIN {X 0,Y 331.2,Z 1216.117,A -85,B 0,C 180,E1 15853.976,E2 15853.976} C_VEL
LIN {X 0,Y 329.707,Z 1224.219,A -85,B 0,C 180,E1 15850.307,E2 15850.307} C_VEL
LIN {X 0,Y 328.81,Z 1230.97,A -85,B 0,C 180,E1 15846.46,E2 15846.46} C_VEL
LIN {X 0,Y 328.444,Z 1235.606,A -85,B 0,C 180,E1 15842.967,E2 15842.967} C_VEL
LIN {X 0,Y 328.347,Z 1239.026,A -85,B 0,C 180,E1 15839.302,E2 15839.302} C_VEL
LIN {X 0,Y 328.427,Z 1241.032,A -85,B 0,C 180,E1 15835.81,E2 15835.81} C_VEL
LIN {X 0,Y 328.746,Z 1241.769,A -85,B 0,C 180,E1 15831.957,E2 15831.957} C_VEL
LIN {X 0,Y 329.505,Z 1241.047,A -85,B 0,C 180,E1 15827.914,E2 15827.914} C_VEL
LIN {X 0,Y 331.025,Z 1238.788,A -85,B 0,C 180,E1 15823.857,E2 15823.857} C_VEL
LIN {X 0,Y 333.645,Z 1234.686,A -85,B 0,C 180,E1 15819.657,E2 15819.657} C_VEL
LIN {X 0,Y 337.571,Z 1228.848,A -85,B 0,C 180,E1 15815.501,E2 15815.501} C_VEL
LIN {X 0,Y 342.672,Z 1221.543,A -85,B 0,C 180,E1 15811.6,E2 15811.6} C_VEL
LIN {X 0,Y 349.471,Z 1212.036,A -85,B 0,C 180,E1 15807.653,E2 15807.653} C_VEL
LIN {X 0,Y 357.445,Z 1200.978,A -85,B 0,C 180,E1 15804.024,E2 15804.024} C_VEL
LIN {X 0,Y 366.848,Z 1187.87,A -85,B 0,C 180,E1 15800.574,E2 15800.574} C_VEL
LIN {X 0,Y 376.723,Z 1173.984,A -85,B 0,C 180,E1 15797.611,E2 15797.611} C_VEL
LIN {X 0,Y 388.402,Z 1157.378,A -85,B 0,C 180,E1 15794.722,E2 15794.722} C_VEL
LIN {X 0,Y 392.478,Z 1151.602,A -85,B 0,C 180,E1 15793.821,E2 15793.821} C_VEL
LIN {X 0,Y 379.431,Z 1166.436,A -85,B 0,C 180,E1 15791.614,E2 15791.614} C_VEL
LIN {X 0,Y 366.41,Z 1183.506,A -85,B 0,C 180,E1 15788.678,E2 15788.678} C_VEL
LIN {X 0,Y 353.263,Z 1204.708,A -85,B 0,C 180,E1 15784.48,E2 15784.48} C_VEL
LIN {X 0,Y 343.388,Z 1224.646,A -85,B 0,C 180,E1 15779.865,E2 15779.865} C_VEL
LIN {X 0,Y 337.152,Z 1240.036,A -85,B 0,C 180,E1 15775.634,E2 15775.634} C_VEL
LIN {X 0,Y 333.117,Z 1252.01,A -85,B 0,C 180,E1 15771.668,E2 15771.668} C_VEL
LIN {X 0,Y 330.496,Z 1261.505,A -85,B 0,C 180,E1 15767.794,E2 15767.794} C_VEL
LIN {X 0,Y 329.005,Z 1268.603,A -85,B 0,C 180,E1 15764.074,E2 15764.074} C_VEL
LIN {X 0,Y 328.341,Z 1273.599,A -85,B 0,C 180,E1 15760.53,E2 15760.53} C_VEL
LIN {X 0,Y 328.198,Z 1276.87,A -85,B 0,C 180,E1 15757.002,E2 15757.002} C_VEL
LIN {X 0,Y 328.302,Z 1278.386,A -85,B 0,C 180,E1 15753.669,E2 15753.669} C_VEL
LIN {X 0,Y 328.436,Z 1278.384,A -85,B 0,C 180,E1 15750.526,E2 15750.526} C_VEL
LIN {X 0,Y 328.465,Z 1276.954,A -85,B 0,C 180,E1 15747.385,E2 15747.385} C_VEL
LIN {X 0,Y 328.426,Z 1273.867,A -85,B 0,C 180,E1 15744.061,E2 15744.061} C_VEL
LIN {X 0,Y 328.443,Z 1269.172,A -85,B 0,C 180,E1 15740.717,E2 15740.717} C_VEL
LIN {X 0,Y 328.767,Z 1262.463,A -85,B 0,C 180,E1 15737.175,E2 15737.175} C_VEL
LIN {X 0,Y 329.581,Z 1253.928,A -85,B 0,C 180,E1 15733.614,E2 15733.614} C_VEL
LIN {X 0,Y 331.056,Z 1243.398,A -85,B 0,C 180,E1 15730.047,E2 15730.047} C_VEL
LIN {X 0,Y 333.451,Z 1230.185,A -85,B 0,C 180,E1 15726.311,E2 15726.311} C_VEL
LIN {X 0,Y 336.826,Z 1214.489,A -85,B 0,C 180,E1 15722.608,E2 15722.608} C_VEL
LIN {X 0,Y 340.865,Z 1197.765,A -85,B 0,C 180,E1 15719.259,E2 15719.259} C_VEL
LIN {X 0,Y 345.879,Z 1178.621,A -85,B 0,C 180,E1 15715.99,E2 15715.99} C_VEL
LIN {X 0,Y 351.813,Z 1156.949,A -85,B 0,C 180,E1 15712.85,E2 15712.85} C_VEL
LIN {X 0,Y 358.579,Z 1132.763,A -85,B 0,C 180,E1 15709.902,E2 15709.902} C_VEL
LIN {X 0,Y 365.309,Z 1108.973,A -85,B 0,C 180,E1 15707.467,E2 15707.467} C_VEL
LIN {X 0,Y 372.823,Z 1082.097,A -85,B 0,C 180,E1 15705.146,E2 15705.146} C_VEL
LIN {X 0,Y 379.895,Z 1056.466,A -85,B 0,C 180,E1 15703.306,E2 15703.306} C_VEL
LIN {X 0,Y 386.45,Z 1031.312,A -85,B 0,C 180,E1 15701.831,E2 15701.831} C_VEL
LIN {X 0,Y 393.303,Z 1002.667,A -85,B 0,C 180,E1 15700.462,E2 15700.462} C_VEL
LIN {X 0,Y 397.463,Z 982.007,A -85,B 0,C 180,E1 15699.632,E2 15699.632} C_VEL
LIN {X 0,Y 390.902,Z 959.475,A -85,B 0,C 180,E1 15697.629,E2 15697.629} C_VEL
LIN {X 0,Y 385.337,Z 934.841,A -85,B 0,C 180,E1 15695.708,E2 15695.708} C_VEL
LIN {X 0,Y 381.268,Z 909.079,A -85,B 0,C 180,E1 15693.914,E2 15693.914} C_VEL
LIN {X 0,Y 380.183,Z 897.909,A -85,B 0,C 180,E1 15693.165,E2 15693.165} C_VEL
LIN {X 0,Y 392.255,Z 843.615,A -85,B 0,C 180,E1 15686.858,E2 15686.858} C_VEL
LIN {X 0,Y 400.328,Z 811.005,A -85,B 0,C 180,E1 15683.088,E2 15683.088} C_VEL
LIN {X 0,Y 402.051,Z 803.575,A -85,B 0,C 180,E1 15682.211,E2 15682.211} C_VEL
LIN {X 0,Y 395.883,Z 786.547,A -85,B 0,C 180,E1 15678.557,E2 15678.557} C_VEL
LIN {X 0,Y 390.046,Z 771.327,A -85,B 0,C 180,E1 15675.006,E2 15675.006} C_VEL
LIN {X 0,Y 384.079,Z 756.572,A -85,B 0,C 180,E1 15671.259,E2 15671.259} C_VEL
LIN {X 0,Y 378.509,Z 743.286,A -85,B 0,C 180,E1 15667.59,E2 15667.59} C_VEL
LIN {X 0,Y 372.831,Z 730.405,A -85,B 0,C 180,E1 15663.69,E2 15663.69} C_VEL
LIN {X 0,Y 367.707,Z 719.182,A -85,B 0,C 180,E1 15660,E2 15660} C_VEL
LIN {X 0,Y 362.971,Z 709.001,A -85,B 0,C 180,E1 15656.367,E2 15656.367} C_VEL
LIN {X 0,Y 358.427,Z 699.388,A -85,B 0,C 180,E1 15652.627,E2 15652.627} C_VEL
LIN {X 0,Y 353.857,Z 690.143,A -85,B 0,C 180,E1 15648.655,E2 15648.655} C_VEL
LIN {X 0,Y 351.058,Z 684.812,A -85,B 0,C 180,E1 15646.158,E2 15646.158} C_VEL
LIN {X 0,Y 349.093,Z 680.767,A -85,B 0,C 180,E1 15644.21,E2 15644.21} C_VEL
LIN {X 0,Y 346.554,Z 675.893,A -85,B 0,C 180,E1 15641.657,E2 15641.657} C_VEL
LIN {X 0,Y 344.303,Z 671.41,A -85,B 0,C 180,E1 15639.239,E2 15639.239} C_VEL
LIN {X 0,Y 342.267,Z 667.419,A -85,B 0,C 180,E1 15636.952,E2 15636.952} C_VEL
LIN {X 0,Y 339.83,Z 663.092,A -85,B 0,C 180,E1 15634.185,E2 15634.185} C_VEL
LIN {X 0,Y 339.163,Z 661.662,A -85,B 0,C 180,E1 15633.281,E2 15633.281} C_VEL
LIN {X 0,Y 337.102,Z 657.937,A -85,B 0,C 180,E1 15630.691,E2 15630.691} C_VEL
LIN {X 0,Y 336.529,Z 656.715,A -85,B 0,C 180,E1 15629.833,E2 15629.833} C_VEL
LIN {X 0,Y 335.596,Z 655.479,A -85,B 0,C 180,E1 15628.573,E2 15628.573} C_VEL
LIN {X 0,Y 337.241,Z 657.267,A -85,B 0,C 180,E1 15627.946,E2 15627.946} C_VEL
LIN {X 0,Y 339.325,Z 661.221,A -85,B 0,C 180,E1 15626.966,E2 15626.966} C_VEL
LIN {X 0,Y 344.848,Z 671.066,A -85,B 0,C 180,E1 15624.556,E2 15624.556} C_VEL
LIN {X 0,Y 351.837,Z 685.286,A -85,B 0,C 180,E1 15621.51,E2 15621.51} C_VEL
LIN {X 0,Y 358.567,Z 700.637,A -85,B 0,C 180,E1 15618.597,E2 15618.597} C_VEL
LIN {X 0,Y 364.242,Z 715.914,A -85,B 0,C 180,E1 15615.986,E2 15615.986} C_VEL
LIN {X 0,Y 369.776,Z 733.417,A -85,B 0,C 180,E1 15613.332,E2 15613.332} C_VEL
LIN {X 0,Y 371.343,Z 739.129,A -85,B 0,C 180,E1 15612.517,E2 15612.517} C_VEL
LIN {X 0,Y 366.448,Z 783.697,A -85,B 0,C 180,E1 15608.568,E2 15608.568} C_VEL
LIN {X 0,Y 361.497,Z 831.902,A -85,B 0,C 180,E1 15604.348,E2 15604.348} C_VEL
LIN {X 0,Y 358.201,Z 870.592,A -85,B 0,C 180,E1 15601.092,E2 15601.092} C_VEL
LIN {X 0,Y 358.561,Z 877.388,A -85,B 0,C 180,E1 15600.897,E2 15600.897} C_VEL
LIN {X 0,Y 353.212,Z 1031.423,A -85,B 0,C 180,E1 15597.86,E2 15597.86} C_VEL
LIN {X 0,Y 352.695,Z 1050.135,A -85,B 0,C 180,E1 15597.32,E2 15597.32} C_VEL
LIN {X 0,Y 351.669,Z 1066.48,A -85,B 0,C 180,E1 15596.572,E2 15596.572} C_VEL
LIN {X 0,Y 350.092,Z 1082.599,A -85,B 0,C 180,E1 15595.545,E2 15595.545} C_VEL
LIN {X 0,Y 348.003,Z 1098.65,A -85,B 0,C 180,E1 15594.202,E2 15594.202} C_VEL
LIN {X 0,Y 345.648,Z 1113.422,A -85,B 0,C 180,E1 15592.625,E2 15592.625} C_VEL
LIN {X 0,Y 343.118,Z 1126.839,A -85,B 0,C 180,E1 15590.823,E2 15590.823} C_VEL
LIN {X 0,Y 340.404,Z 1139.695,A -85,B 0,C 180,E1 15588.671,E2 15588.671} C_VEL
LIN {X 0,Y 337.843,Z 1150.927,A -85,B 0,C 180,E1 15586.327,E2 15586.327} C_VEL
LIN {X 0,Y 335.531,Z 1160.546,A -85,B 0,C 180,E1 15583.79,E2 15583.79} C_VEL
LIN {X 0,Y 333.563,Z 1168.609,A -85,B 0,C 180,E1 15581.058,E2 15581.058} C_VEL
LIN {X 0,Y 332.027,Z 1175.113,A -85,B 0,C 180,E1 15578.134,E2 15578.134} C_VEL
LIN {X 0,Y 330.998,Z 1179.688,A -85,B 0,C 180,E1 15575.197,E2 15575.197} C_VEL
LIN {X 0,Y 330.395,Z 1182.605,A -85,B 0,C 180,E1 15572.079,E2 15572.079} C_VEL
LIN {X 0,Y 330.22,Z 1183.723,A -85,B 0,C 180,E1 15568.957,E2 15568.957} C_VEL
LIN {X 0,Y 330.443,Z 1183.042,A -85,B 0,C 180,E1 15565.833,E2 15565.833} C_VEL
LIN {X 0,Y 331.098,Z 1180.48,A -85,B 0,C 180,E1 15562.711,E2 15562.711} C_VEL
LIN {X 0,Y 332.195,Z 1176.314,A -85,B 0,C 180,E1 15559.769,E2 15559.769} C_VEL
LIN {X 0,Y 333.818,Z 1170.305,A -85,B 0,C 180,E1 15556.839,E2 15556.839} C_VEL
LIN {X 0,Y 335.917,Z 1162.448,A -85,B 0,C 180,E1 15554.038,E2 15554.038} C_VEL
LIN {X 0,Y 338.447,Z 1152.833,A -85,B 0,C 180,E1 15551.391,E2 15551.391} C_VEL
LIN {X 0,Y 341.145,Z 1142.072,A -85,B 0,C 180,E1 15549.046,E2 15549.046} C_VEL
LIN {X 0,Y 343.977,Z 1129.628,A -85,B 0,C 180,E1 15546.892,E2 15546.892} C_VEL
LIN {X 0,Y 346.741,Z 1116.076,A -85,B 0,C 180,E1 15545.008,E2 15545.008} C_VEL
LIN {X 0,Y 349.305,Z 1101.496,A -85,B 0,C 180,E1 15543.384,E2 15543.384} C_VEL
LIN {X 0,Y 351.557,Z 1085.667,A -85,B 0,C 180,E1 15542.01,E2 15542.01} C_VEL
LIN {X 0,Y 353.333,Z 1069.149,A -85,B 0,C 180,E1 15540.918,E2 15540.918} C_VEL
LIN {X 0,Y 354.57,Z 1051.861,A -85,B 0,C 180,E1 15540.09,E2 15540.09} C_VEL
LIN {X 0,Y 355.162,Z 1033.967,A -85,B 0,C 180,E1 15539.545,E2 15539.545} C_VEL
LIN {X 0,Y 357.606,Z 958.724,A -85,B 0,C 180,E1 15538.041,E2 15538.041} C_VEL
LIN {X 0,Y 360.673,Z 874.851,A -85,B 0,C 180,E1 15536.397,E2 15536.397} C_VEL
LIN {X 0,Y 360.241,Z 869.608,A -85,B 0,C 180,E1 15536.183,E2 15536.183} C_VEL
LIN {X 0,Y 363.024,Z 839.755,A -85,B 0,C 180,E1 15533.637,E2 15533.637} C_VEL
LIN {X 0,Y 364.957,Z 840.157,A -85,B 0,C 180,E1 15533.324,E2 15533.324} C_VEL
LIN {X 0,Y 368.028,Z 838.505,A -85,B 0,C 180,E1 15532.951,E2 15532.951} C_VEL
LIN {X 0,Y 372.409,Z 833.642,A -85,B 0,C 180,E1 15532.543,E2 15532.543} C_VEL
LIN {X 0,Y 377.49,Z 830.98,A -85,B 0,C 180,E1 15531.937,E2 15531.937} C_VEL
LIN {X 0,Y 382.159,Z 826.486,A -85,B 0,C 180,E1 15531.484,E2 15531.484} C_VEL
LIN {X 0,Y 383.44,Z 825.487,A -85,B 0,C 180,E1 15531.35,E2 15531.35} C_VEL
LIN {X 0,Y 388.71,Z 822.1,A -85,B 0,C 180,E1 15530.77,E2 15530.77} C_VEL
LIN {X 0,Y 393.446,Z 817.778,A -85,B 0,C 180,E1 15530.317,E2 15530.317} C_VEL
LIN {X 0,Y 393.598,Z 817.697,A -85,B 0,C 180,E1 15530.3,E2 15530.3} C_VEL
LIN {X 0,Y 394.877,Z 817.962,A -85,B 0,C 180,E1 15530.115,E2 15530.115} C_VEL
LIN {X 0,Y 396.088,Z 820.425,A -85,B 0,C 180,E1 15529.847,E2 15529.847} C_VEL
LIN {X 0,Y 396.373,Z 825.055,A -85,B 0,C 180,E1 15529.609,E2 15529.609} C_VEL
LIN {X 0,Y 394.026,Z 840.58,A -85,B 0,C 180,E1 15529.249,E2 15529.249} C_VEL
LIN {X 0,Y 377.082,Z 981.788,A -85,B 0,C 180,E1 15525.149,E2 15525.149} C_VEL
LIN {X 0,Y 374.229,Z 1006.359,A -85,B 0,C 180,E1 15524.245,E2 15524.245} C_VEL
LIN {X 0,Y 370.653,Z 1030.163,A -85,B 0,C 180,E1 15523.093,E2 15523.093} C_VEL
LIN {X 0,Y 366.57,Z 1052.557,A -85,B 0,C 180,E1 15521.725,E2 15521.725} C_VEL
LIN {X 0,Y 361.902,Z 1074.576,A -85,B 0,C 180,E1 15520.072,E2 15520.072} C_VEL
LIN {X 0,Y 356.901,Z 1095.503,A -85,B 0,C 180,E1 15518.152,E2 15518.152} C_VEL
LIN {X 0,Y 351.839,Z 1114.827,A -85,B 0,C 180,E1 15516.035,E2 15516.035} C_VEL
LIN {X 0,Y 346.312,Z 1134.498,A -85,B 0,C 180,E1 15513.468,E2 15513.468} C_VEL
LIN {X 0,Y 341.365,Z 1151.478,A -85,B 0,C 180,E1 15510.837,E2 15510.837} C_VEL
LIN {X 0,Y 336.455,Z 1167.929,A -85,B 0,C 180,E1 15507.813,E2 15507.813} C_VEL
LIN {X 0,Y 332.266,Z 1182.016,A -85,B 0,C 180,E1 15504.727,E2 15504.727} C_VEL
LIN {X 0,Y 328.431,Z 1195.456,A -85,B 0,C 180,E1 15501.241,E2 15501.241} C_VEL
LIN {X 0,Y 325.454,Z 1206.862,A -85,B 0,C 180,E1 15497.708,E2 15497.708} C_VEL
LIN {X 0,Y 323.174,Z 1216.815,A -85,B 0,C 180,E1 15493.965,E2 15493.965} C_VEL
LIN {X 0,Y 321.668,Z 1224.895,A -85,B 0,C 180,E1 15490.206,E2 15490.206} C_VEL
LIN {X 0,Y 320.785,Z 1231.623,A -85,B 0,C 180,E1 15486.263,E2 15486.263} C_VEL
LIN {X 0,Y 320.432,Z 1236.25,A -85,B 0,C 180,E1 15482.683,E2 15482.683} C_VEL
LIN {X 0,Y 320.358,Z 1239.656,A -85,B 0,C 180,E1 15478.927,E2 15478.927} C_VEL
LIN {X 0,Y 320.471,Z 1241.747,A -85,B 0,C 180,E1 15475.168,E2 15475.168} C_VEL
LIN {X 0,Y 320.845,Z 1242.402,A -85,B 0,C 180,E1 15471.397,E2 15471.397} C_VEL
LIN {X 0,Y 321.734,Z 1241.699,A -85,B 0,C 180,E1 15467.252,E2 15467.252} C_VEL
LIN {X 0,Y 323.461,Z 1239.488,A -85,B 0,C 180,E1 15463.108,E2 15463.108} C_VEL
LIN {X 0,Y 326.553,Z 1235.264,A -85,B 0,C 180,E1 15458.631,E2 15458.631} C_VEL
LIN {X 0,Y 330.929,Z 1229.439,A -85,B 0,C 180,E1 15454.401,E2 15454.401} C_VEL
LIN {X 0,Y 336.807,Z 1221.848,A -85,B 0,C 180,E1 15450.279,E2 15450.279} C_VEL
LIN {X 0,Y 344.264,Z 1212.376,A -85,B 0,C 180,E1 15446.307,E2 15446.307} C_VEL
LIN {X 0,Y 352.909,Z 1201.419,A -85,B 0,C 180,E1 15442.676,E2 15442.676} C_VEL
LIN {X 0,Y 362.568,Z 1189.13,A -85,B 0,C 180,E1 15439.395,E2 15439.395} C_VEL
LIN {X 0,Y 374.243,Z 1174.183,A -85,B 0,C 180,E1 15436.17,E2 15436.17} C_VEL
LIN {X 0,Y 383.972,Z 1161.619,A -85,B 0,C 180,E1 15433.897,E2 15433.897} C_VEL
LIN {X 0,Y 369.495,Z 1177.205,A -85,B 0,C 180,E1 15431.324,E2 15431.324} C_VEL
LIN {X 0,Y 355.785,Z 1194.56,A -85,B 0,C 180,E1 15427.988,E2 15427.988} C_VEL
LIN {X 0,Y 343.146,Z 1214.235,A -85,B 0,C 180,E1 15423.619,E2 15423.619} C_VEL
LIN {X 0,Y 334.007,Z 1231.911,A -85,B 0,C 180,E1 15419.012,E2 15419.012} C_VEL
LIN {X 0,Y 328.074,Z 1245.8,A -85,B 0,C 180,E1 15414.682,E2 15414.682} C_VEL
LIN {X 0,Y 324.261,Z 1256.547,A -85,B 0,C 180,E1 15410.583,E2 15410.583} C_VEL
LIN {X 0,Y 321.928,Z 1264.847,A -85,B 0,C 180,E1 15406.606,E2 15406.606} C_VEL
LIN {X 0,Y 320.7,Z 1270.901,A -85,B 0,C 180,E1 15402.792,E2 15402.792} C_VEL
LIN {X 0,Y 320.226,Z 1274.947,A -85,B 0,C 180,E1 15399.165,E2 15399.165} C_VEL
LIN {X 0,Y 320.236,Z 1277.294,A -85,B 0,C 180,E1 15395.557,E2 15395.557} C_VEL
LIN {X 0,Y 320.397,Z 1277.934,A -85,B 0,C 180,E1 15392.149,E2 15392.149} C_VEL
LIN {X 0,Y 320.503,Z 1277.091,A -85,B 0,C 180,E1 15388.93,E2 15388.93} C_VEL
LIN {X 0,Y 320.48,Z 1274.812,A -85,B 0,C 180,E1 15385.708,E2 15385.708} C_VEL
LIN {X 0,Y 320.441,Z 1270.825,A -85,B 0,C 180,E1 15382.292,E2 15382.292} C_VEL
LIN {X 0,Y 320.603,Z 1264.865,A -85,B 0,C 180,E1 15378.671,E2 15378.671} C_VEL
LIN {X 0,Y 321.197,Z 1257.086,A -85,B 0,C 180,E1 15375.029,E2 15375.029} C_VEL
LIN {X 0,Y 322.409,Z 1247.331,A -85,B 0,C 180,E1 15371.374,E2 15371.374} C_VEL
LIN {X 0,Y 324.509,Z 1234.971,A -85,B 0,C 180,E1 15367.541,E2 15367.541} C_VEL
LIN {X 0,Y 327.584,Z 1220.207,A -85,B 0,C 180,E1 15363.734,E2 15363.734} C_VEL
LIN {X 0,Y 331.294,Z 1204.668,A -85,B 0,C 180,E1 15360.335,E2 15360.335} C_VEL
LIN {X 0,Y 336.202,Z 1185.829,A -85,B 0,C 180,E1 15356.826,E2 15356.826} C_VEL
LIN {X 0,Y 342.216,Z 1164.094,A -85,B 0,C 180,E1 15353.416,E2 15353.416} C_VEL
LIN {X 0,Y 349.018,Z 1140.382,A -85,B 0,C 180,E1 15350.296,E2 15350.296} C_VEL
LIN {X 0,Y 356.452,Z 1114.599,A -85,B 0,C 180,E1 15347.469,E2 15347.469} C_VEL
LIN {X 0,Y 363.451,Z 1090.398,A -85,B 0,C 180,E1 15345.232,E2 15345.232} C_VEL
LIN {X 0,Y 370.94,Z 1063.908,A -85,B 0,C 180,E1 15343.189,E2 15343.189} C_VEL
LIN {X 0,Y 378.017,Z 1038.044,A -85,B 0,C 180,E1 15341.538,E2 15341.538} C_VEL
LIN {X 0,Y 384.736,Z 1011.66,A -85,B 0,C 180,E1 15340.179,E2 15340.179} C_VEL
LIN {X 0,Y 390.705,Z 984.299,A -85,B 0,C 180,E1 15339.018,E2 15339.018} C_VEL
LIN {X 0,Y 385.065,Z 964.209,A -85,B 0,C 180,E1 15337.18,E2 15337.18} C_VEL
LIN {X 0,Y 379.94,Z 940.905,A -85,B 0,C 180,E1 15335.286,E2 15335.286} C_VEL
LIN {X 0,Y 375.956,Z 916.479,A -85,B 0,C 180,E1 15333.53,E2 15333.53} C_VEL
LIN {X 0,Y 373.918,Z 895.925,A -85,B 0,C 180,E1 15332.151,E2 15332.151} C_VEL
LIN {X 0,Y 385.503,Z 846.221,A -85,B 0,C 180,E1 15326.329,E2 15326.329} C_VEL
LIN {X 0,Y 393.724,Z 813.775,A -85,B 0,C 180,E1 15322.549,E2 15322.549} C_VEL
LIN {X 0,Y 395.33,Z 807.079,A -85,B 0,C 180,E1 15321.749,E2 15321.749} C_VEL
LIN {X 0,Y 389.326,Z 790.379,A -85,B 0,C 180,E1 15318.105,E2 15318.105} C_VEL
LIN {X 0,Y 383.291,Z 774.579,A -85,B 0,C 180,E1 15314.349,E2 15314.349} C_VEL
LIN {X 0,Y 377.171,Z 759.296,A -85,B 0,C 180,E1 15310.386,E2 15310.386} C_VEL
LIN {X 0,Y 371.272,Z 745.322,A -85,B 0,C 180,E1 15306.425,E2 15306.425} C_VEL
LIN {X 0,Y 365.944,Z 733.183,A -85,B 0,C 180,E1 15302.662,E2 15302.662} C_VEL
LIN {X 0,Y 360.7,Z 721.616,A -85,B 0,C 180,E1 15298.729,E2 15298.729} C_VEL
LIN {X 0,Y 355.962,Z 711.661,A -85,B 0,C 180,E1 15295.004,E2 15295.004} C_VEL
LIN {X 0,Y 351.625,Z 702.58,A -85,B 0,C 180,E1 15291.332,E2 15291.332} C_VEL
LIN {X 0,Y 347.963,Z 695.139,A -85,B 0,C 180,E1 15288.059,E2 15288.059} C_VEL
LIN {X 0,Y 345.516,Z 690.318,A -85,B 0,C 180,E1 15285.79,E2 15285.79} C_VEL
LIN {X 0,Y 343.532,Z 686.307,A -85,B 0,C 180,E1 15283.832,E2 15283.832} C_VEL
LIN {X 0,Y 341.359,Z 681.948,A -85,B 0,C 180,E1 15281.558,E2 15281.558} C_VEL
LIN {X 0,Y 339.126,Z 677.462,A -85,B 0,C 180,E1 15279.098,E2 15279.098} C_VEL
LIN {X 0,Y 336.524,Z 672.536,A -85,B 0,C 180,E1 15276.166,E2 15276.166} C_VEL
LIN {X 0,Y 334.541,Z 668.59,A -85,B 0,C 180,E1 15273.715,E2 15273.715} C_VEL
LIN {X 0,Y 331.949,Z 663.819,A -85,B 0,C 180,E1 15270.396,E2 15270.396} C_VEL
LIN {X 0,Y 330.838,Z 662.109,A -85,B 0,C 180,E1 15268.881,E2 15268.881} C_VEL
LIN {X 0,Y 332.472,Z 663.438,A -85,B 0,C 180,E1 15268.306,E2 15268.306} C_VEL
LIN {X 0,Y 338.979,Z 675.458,A -85,B 0,C 180,E1 15265.299,E2 15265.299} C_VEL
LIN {X 0,Y 344.297,Z 686.203,A -85,B 0,C 180,E1 15262.838,E2 15262.838} C_VEL
LIN {X 0,Y 350.914,Z 700.786,A -85,B 0,C 180,E1 15259.912,E2 15259.912} C_VEL
LIN {X 0,Y 357.407,Z 717.741,A -85,B 0,C 180,E1 15256.897,E2 15256.897} C_VEL
LIN {X 0,Y 363.077,Z 735.784,A -85,B 0,C 180,E1 15254.046,E2 15254.046} C_VEL
LIN {X 0,Y 364.853,Z 742.495,A -85,B 0,C 180,E1 15253.081,E2 15253.081} C_VEL
LIN {X 0,Y 359.533,Z 788.828,A -85,B 0,C 180,E1 15248.938,E2 15248.938} C_VEL
LIN {X 0,Y 354.325,Z 838.725,A -85,B 0,C 180,E1 15244.553,E2 15244.553} C_VEL
LIN {X 0,Y 351.437,Z 871.516,A -85,B 0,C 180,E1 15241.773,E2 15241.773} C_VEL
LIN {X 0,Y 351.781,Z 878.26,A -85,B 0,C 180,E1 15241.575,E2 15241.575} C_VEL
LIN {X 0,Y 346.236,Z 1031.798,A -85,B 0,C 180,E1 15238.498,E2 15238.498} C_VEL
LIN {X 0,Y 345.697,Z 1050.673,A -85,B 0,C 180,E1 15237.95,E2 15237.95} C_VEL
LIN {X 0,Y 344.583,Z 1067.72,A -85,B 0,C 180,E1 15237.157,E2 15237.157} C_VEL
LIN {X 0,Y 342.915,Z 1084.03,A -85,B 0,C 180,E1 15236.092,E2 15236.092} C_VEL
LIN {X 0,Y 340.735,Z 1100.066,A -85,B 0,C 180,E1 15234.716,E2 15234.716} C_VEL
LIN {X 0,Y 338.341,Z 1114.477,A -85,B 0,C 180,E1 15233.142,E2 15233.142} C_VEL
LIN {X 0,Y 335.715,Z 1127.873,A -85,B 0,C 180,E1 15231.304,E2 15231.304} C_VEL
LIN {X 0,Y 332.896,Z 1140.716,A -85,B 0,C 180,E1 15229.108,E2 15229.108} C_VEL
LIN {X 0,Y 330.233,Z 1151.937,A -85,B 0,C 180,E1 15226.714,E2 15226.714} C_VEL
LIN {X 0,Y 327.825,Z 1161.542,A -85,B 0,C 180,E1 15224.12,E2 15224.12} C_VEL
LIN {X 0,Y 325.772,Z 1169.597,A -85,B 0,C 180,E1 15221.326,E2 15221.326} C_VEL
LIN {X 0,Y 324.166,Z 1176.093,A -85,B 0,C 180,E1 15218.333,E2 15218.333} C_VEL
LIN {X 0,Y 323.089,Z 1180.657,A -85,B 0,C 180,E1 15215.325,E2 15215.325} C_VEL
LIN {X 0,Y 322.458,Z 1183.567,A -85,B 0,C 180,E1 15212.13,E2 15212.13} C_VEL
LIN {X 0,Y 322.278,Z 1184.678,A -85,B 0,C 180,E1 15208.931,E2 15208.931} C_VEL
LIN {X 0,Y 322.515,Z 1183.987,A -85,B 0,C 180,E1 15205.73,E2 15205.73} C_VEL
LIN {X 0,Y 323.208,Z 1181.417,A -85,B 0,C 180,E1 15202.532,E2 15202.532} C_VEL
LIN {X 0,Y 324.363,Z 1177.244,A -85,B 0,C 180,E1 15199.519,E2 15199.519} C_VEL
LIN {X 0,Y 326.068,Z 1171.224,A -85,B 0,C 180,E1 15196.521,E2 15196.521} C_VEL
LIN {X 0,Y 328.211,Z 1163.561,A -85,B 0,C 180,E1 15193.721,E2 15193.721} C_VEL
LIN {X 0,Y 330.724,Z 1154.405,A -85,B 0,C 180,E1 15191.123,E2 15191.123} C_VEL
LIN {X 0,Y 333.505,Z 1143.783,A -85,B 0,C 180,E1 15188.727,E2 15188.727} C_VEL
LIN {X 0,Y 336.433,Z 1131.563,A -85,B 0,C 180,E1 15186.529,E2 15186.529} C_VEL
LIN {X 0,Y 339.283,Z 1118.208,A -85,B 0,C 180,E1 15184.607,E2 15184.607} C_VEL
LIN {X 0,Y 341.932,Z 1103.878,A -85,B 0,C 180,E1 15182.951,E2 15182.951} C_VEL
LIN {X 0,Y 344.274,Z 1088.58,A -85,B 0,C 180,E1 15181.553,E2 15181.553} C_VEL
LIN {X 0,Y 346.121,Z 1072.672,A -85,B 0,C 180,E1 15180.442,E2 15180.442} C_VEL
LIN {X 0,Y 347.503,Z 1055.151,A -85,B 0,C 180,E1 15179.549,E2 15179.549} C_VEL
LIN {X 0,Y 348.232,Z 1037.451,A -85,B 0,C 180,E1 15178.955,E2 15178.955} C_VEL
LIN {X 0,Y 349.967,Z 981.372,A -85,B 0,C 180,E1 15177.794,E2 15177.794} C_VEL
LIN {X 0,Y 354.002,Z 875.731,A -85,B 0,C 180,E1 15175.693,E2 15175.693} C_VEL
LIN {X 0,Y 353.598,Z 870.308,A -85,B 0,C 180,E1 15175.459,E2 15175.459} C_VEL
LIN {X 0,Y 355.23,Z 854.321,A -85,B 0,C 180,E1 15174.062,E2 15174.062} C_VEL
LIN {X 0,Y 357.003,Z 854.678,A -85,B 0,C 180,E1 15173.772,E2 15173.772} C_VEL
LIN {X 0,Y 360.098,Z 853.045,A -85,B 0,C 180,E1 15173.388,E2 15173.388} C_VEL
LIN {X 0,Y 364.145,Z 848.63,A -85,B 0,C 180,E1 15173.01,E2 15173.01} C_VEL
LIN {X 0,Y 364.966,Z 847.762,A -85,B 0,C 180,E1 15172.932,E2 15172.932} C_VEL
LIN {X 0,Y 369.026,Z 845.866,A -85,B 0,C 180,E1 15172.434,E2 15172.434} C_VEL
LIN {X 0,Y 373.688,Z 841.59,A -85,B 0,C 180,E1 15171.967,E2 15171.967} C_VEL
LIN {X 0,Y 375.283,Z 840.073,A -85,B 0,C 180,E1 15171.812,E2 15171.812} C_VEL
LIN {X 0,Y 380.481,Z 836.881,A -85,B 0,C 180,E1 15171.234,E2 15171.234} C_VEL
LIN {X 0,Y 385.568,Z 832.203,A -85,B 0,C 180,E1 15170.744,E2 15170.744} C_VEL
LIN {X 0,Y 391.473,Z 828.202,A -85,B 0,C 180,E1 15170.124,E2 15170.124} C_VEL
LIN {X 0,Y 396.046,Z 824.212,A -85,B 0,C 180,E1 15169.688,E2 15169.688} C_VEL
LIN {X 0,Y 394.026,Z 840.58,A -85,B 0,C 180,E1 15169.249,E2 15169.249} C_VEL
LIN {X 0,Y 392.342,Z 848.126,A -85,B 0,C 180,E1 15169.142,E2 15169.142} C_VEL
LIN {X 0,Y 385.102,Z 868.1,A -85,B 0,C 180,E1 15169.192,E2 15169.192} C_VEL
LIN {X 0,Y 383.695,Z 874.566,A -85,B 0,C 180,E1 15169.08,E2 15169.08} C_VEL
LIN {X 0,Y 370.269,Z 983.611,A -85,B 0,C 180,E1 15165.777,E2 15165.777} C_VEL
LIN {X 0,Y 367.241,Z 1008.443,A -85,B 0,C 180,E1 15164.831,E2 15164.831} C_VEL
LIN {X 0,Y 363.558,Z 1031.995,A -85,B 0,C 180,E1 15163.656,E2 15163.656} C_VEL
LIN {X 0,Y 359.336,Z 1054.365,A -85,B 0,C 180,E1 15162.252,E2 15162.252} C_VEL
LIN {X 0,Y 354.726,Z 1075.508,A -85,B 0,C 180,E1 15160.628,E2 15160.628} C_VEL
LIN {X 0,Y 349.412,Z 1097.131,A -85,B 0,C 180,E1 15158.597,E2 15158.597} C_VEL
LIN {X 0,Y 344.06,Z 1116.939,A -85,B 0,C 180,E1 15156.36,E2 15156.36} C_VEL
LIN {X 0,Y 338.661,Z 1135.62,A -85,B 0,C 180,E1 15153.85,E2 15153.85} C_VEL
LIN {X 0,Y 333.413,Z 1153.149,A -85,B 0,C 180,E1 15151.053,E2 15151.053} C_VEL
LIN {X 0,Y 328.428,Z 1169.476,A -85,B 0,C 180,E1 15147.96,E2 15147.96} C_VEL
LIN {X 0,Y 323.974,Z 1184.169,A -85,B 0,C 180,E1 15144.624,E2 15144.624} C_VEL
LIN {X 0,Y 320.32,Z 1196.739,A -85,B 0,C 180,E1 15141.229,E2 15141.229} C_VEL
LIN {X 0,Y 317.325,Z 1208.023,A -85,B 0,C 180,E1 15137.608,E2 15137.608} C_VEL
LIN {X 0,Y 315.051,Z 1217.917,A -85,B 0,C 180,E1 15133.77,E2 15133.77} C_VEL
LIN {X 0,Y 313.574,Z 1225.891,A -85,B 0,C 180,E1 15129.915,E2 15129.915} C_VEL
LIN {X 0,Y 312.731,Z 1232.51,A -85,B 0,C 180,E1 15125.872,E2 15125.872} C_VEL
LIN {X 0,Y 312.406,Z 1237.298,A -85,B 0,C 180,E1 15122.018,E2 15122.018} C_VEL
LIN {X 0,Y 312.374,Z 1240.527,A -85,B 0,C 180,E1 15118.166,E2 15118.166} C_VEL
LIN {X 0,Y 312.554,Z 1242.51,A -85,B 0,C 180,E1 15114.237,E2 15114.237} C_VEL
LIN {X 0,Y 313.007,Z 1243.057,A -85,B 0,C 180,E1 15110.438,E2 15110.438} C_VEL
LIN {X 0,Y 314.148,Z 1242.204,A -85,B 0,C 180,E1 15106.121,E2 15106.121} C_VEL
LIN {X 0,Y 316.284,Z 1239.776,A -85,B 0,C 180,E1 15101.761,E2 15101.761} C_VEL
LIN {X 0,Y 319.75,Z 1235.682,A -85,B 0,C 180,E1 15097.379,E2 15097.379} C_VEL
LIN {X 0,Y 324.92,Z 1229.592,A -85,B 0,C 180,E1 15092.906,E2 15092.906} C_VEL
LIN {X 0,Y 332.017,Z 1221.342,A -85,B 0,C 180,E1 15088.463,E2 15088.463} C_VEL
LIN {X 0,Y 340.458,Z 1211.598,A -85,B 0,C 180,E1 15084.443,E2 15084.443} C_VEL
LIN {X 0,Y 350.449,Z 1200.016,A -85,B 0,C 180,E1 15080.698,E2 15080.698} C_VEL
LIN {X 0,Y 361.566,Z 1187.058,A -85,B 0,C 180,E1 15077.349,E2 15077.349} C_VEL
LIN {X 0,Y 374.849,Z 1171.59,A -85,B 0,C 180,E1 15074.148,E2 15074.148} C_VEL
LIN {X 0,Y 375.449,Z 1170.909,A -85,B 0,C 180,E1 15073.989,E2 15073.989} C_VEL
LIN {X 0,Y 361.335,Z 1185.213,A -85,B 0,C 180,E1 15071.406,E2 15071.406} C_VEL
LIN {X 0,Y 347.11,Z 1202.12,A -85,B 0,C 180,E1 15067.85,E2 15067.85} C_VEL
LIN {X 0,Y 334.147,Z 1221.07,A -85,B 0,C 180,E1 15063.205,E2 15063.205} C_VEL
LIN {X 0,Y 324.992,Z 1237.707,A -85,B 0,C 180,E1 15058.366,E2 15058.366} C_VEL
LIN {X 0,Y 319.363,Z 1250.043,A -85,B 0,C 180,E1 15054.02,E2 15054.02} C_VEL
LIN {X 0,Y 315.714,Z 1259.742,A -85,B 0,C 180,E1 15049.811,E2 15049.811} C_VEL
LIN {X 0,Y 313.55,Z 1267.1,A -85,B 0,C 180,E1 15045.73,E2 15045.73} C_VEL
LIN {X 0,Y 312.505,Z 1272.308,A -85,B 0,C 180,E1 15041.819,E2 15041.819} C_VEL
LIN {X 0,Y 312.2,Z 1275.583,A -85,B 0,C 180,E1 15038.103,E2 15038.103} C_VEL
LIN {X 0,Y 312.29,Z 1277.139,A -85,B 0,C 180,E1 15034.594,E2 15034.594} C_VEL
LIN {X 0,Y 312.464,Z 1277.198,A -85,B 0,C 180,E1 15031.286,E2 15031.286} C_VEL
LIN {X 0,Y 312.539,Z 1275.833,A -85,B 0,C 180,E1 15027.986,E2 15027.986} C_VEL
LIN {X 0,Y 312.502,Z 1273.014,A -85,B 0,C 180,E1 15024.678,E2 15024.678} C_VEL
LIN {X 0,Y 312.491,Z 1268.431,A -85,B 0,C 180,E1 15021.168,E2 15021.168} C_VEL
LIN {X 0,Y 312.753,Z 1262.196,A -85,B 0,C 180,E1 15017.634,E2 15017.634} C_VEL
LIN {X 0,Y 313.572,Z 1253.323,A -85,B 0,C 180,E1 15013.7,E2 15013.7} C_VEL
LIN {X 0,Y 315.064,Z 1242.885,A -85,B 0,C 180,E1 15009.95,E2 15009.95} C_VEL
LIN {X 0,Y 317.626,Z 1229.296,A -85,B 0,C 180,E1 15005.913,E2 15005.913} C_VEL
LIN {X 0,Y 320.981,Z 1214.381,A -85,B 0,C 180,E1 15002.214,E2 15002.214} C_VEL
LIN {X 0,Y 325.201,Z 1197.721,A -85,B 0,C 180,E1 14998.696,E2 14998.696} C_VEL
LIN {X 0,Y 330.76,Z 1177.512,A -85,B 0,C 180,E1 14995.089,E2 14995.089} C_VEL
LIN {X 0,Y 337.259,Z 1154.999,A -85,B 0,C 180,E1 14991.714,E2 14991.714} C_VEL
LIN {X 0,Y 344.406,Z 1130.717,A -85,B 0,C 180,E1 14988.667,E2 14988.667} C_VEL
LIN {X 0,Y 351.716,Z 1106.076,A -85,B 0,C 180,E1 14986.083,E2 14986.083} C_VEL
LIN {X 0,Y 359.632,Z 1079.142,A -85,B 0,C 180,E1 14983.711,E2 14983.711} C_VEL
LIN {X 0,Y 367.034,Z 1053.543,A -85,B 0,C 180,E1 14981.838,E2 14981.838} C_VEL
LIN {X 0,Y 374.134,Z 1027.488,A -85,B 0,C 180,E1 14980.286,E2 14980.286} C_VEL
LIN {X 0,Y 381.08,Z 999.596,A -85,B 0,C 180,E1 14978.93,E2 14978.93} C_VEL
LIN {X 0,Y 383.888,Z 986.252,A -85,B 0,C 180,E1 14978.352,E2 14978.352} C_VEL
LIN {X 0,Y 377.746,Z 962.665,A -85,B 0,C 180,E1 14976.177,E2 14976.177} C_VEL
LIN {X 0,Y 373.31,Z 940.807,A -85,B 0,C 180,E1 14974.39,E2 14974.39} C_VEL
LIN {X 0,Y 369.51,Z 914.622,A -85,B 0,C 180,E1 14972.489,E2 14972.489} C_VEL
LIN {X 0,Y 367.806,Z 893.811,A -85,B 0,C 180,E1 14971.098,E2 14971.098} C_VEL
LIN {X 0,Y 378.72,Z 849.033,A -85,B 0,C 180,E1 14965.809,E2 14965.809} C_VEL
LIN {X 0,Y 387.156,Z 816.541,A -85,B 0,C 180,E1 14961.993,E2 14961.993} C_VEL
LIN {X 0,Y 388.619,Z 810.608,A -85,B 0,C 180,E1 14961.271,E2 14961.271} C_VEL
LIN {X 0,Y 382.56,Z 793.581,A -85,B 0,C 180,E1 14957.492,E2 14957.492} C_VEL
LIN {X 0,Y 376.519,Z 777.778,A -85,B 0,C 180,E1 14953.671,E2 14953.671} C_VEL
LIN {X 0,Y 370.632,Z 763.046,A -85,B 0,C 180,E1 14949.786,E2 14949.786} C_VEL
LIN {X 0,Y 365.071,Z 749.866,A -85,B 0,C 180,E1 14945.974,E2 14945.974} C_VEL
LIN {X 0,Y 359.916,Z 737.966,A -85,B 0,C 180,E1 14942.229,E2 14942.229} C_VEL
LIN {X 0,Y 354.691,Z 726.391,A -85,B 0,C 180,E1 14938.223,E2 14938.223} C_VEL
LIN {X 0,Y 349.98,Z 716.317,A -85,B 0,C 180,E1 14934.426,E2 14934.426} C_VEL
LIN {X 0,Y 345.503,Z 706.7,A -85,B 0,C 180,E1 14930.505,E2 14930.505} C_VEL
LIN {X 0,Y 342.337,Z 700.542,A -85,B 0,C 180,E1 14927.689,E2 14927.689} C_VEL
LIN {X 0,Y 340.307,Z 696.39,A -85,B 0,C 180,E1 14925.711,E2 14925.711} C_VEL
LIN {X 0,Y 338.068,Z 691.949,A -85,B 0,C 180,E1 14923.505,E2 14923.505} C_VEL
LIN {X 0,Y 335.929,Z 687.664,A -85,B 0,C 180,E1 14921.249,E2 14921.249} C_VEL
LIN {X 0,Y 333.682,Z 683.173,A -85,B 0,C 180,E1 14918.728,E2 14918.728} C_VEL
LIN {X 0,Y 331.309,Z 678.528,A -85,B 0,C 180,E1 14915.956,E2 14915.956} C_VEL
LIN {X 0,Y 328.82,Z 673.757,A -85,B 0,C 180,E1 14912.862,E2 14912.862} C_VEL
LIN {X 0,Y 326.495,Z 669.146,A -85,B 0,C 180,E1 14909.648,E2 14909.648} C_VEL
LIN {X 0,Y 326.141,Z 668.737,A -85,B 0,C 180,E1 14909.203,E2 14909.203} C_VEL
LIN {X 0,Y 327.813,Z 669.72,A -85,B 0,C 180,E1 14908.649,E2 14908.649} C_VEL
LIN {X 0,Y 334.606,Z 682.357,A -85,B 0,C 180,E1 14905.405,E2 14905.405} C_VEL
LIN {X 0,Y 341.249,Z 696.447,A -85,B 0,C 180,E1 14902.237,E2 14902.237} C_VEL
LIN {X 0,Y 347.253,Z 710.804,A -85,B 0,C 180,E1 14899.401,E2 14899.401} C_VEL
LIN {X 0,Y 353.151,Z 727.31,A -85,B 0,C 180,E1 14896.526,E2 14896.526} C_VEL
LIN {X 0,Y 358.065,Z 744.098,A -85,B 0,C 180,E1 14893.907,E2 14893.907} C_VEL
LIN {X 0,Y 358.374,Z 745.858,A -85,B 0,C 180,E1 14893.669,E2 14893.669} C_VEL
LIN {X 0,Y 352.904,Z 792.25,A -85,B 0,C 180,E1 14889.497,E2 14889.497} C_VEL
LIN {X 0,Y 347.547,Z 841.494,A -85,B 0,C 180,E1 14885.124,E2 14885.124} C_VEL
LIN {X 0,Y 344.727,Z 872.472,A -85,B 0,C 180,E1 14882.479,E2 14882.479} C_VEL
LIN {X 0,Y 345.052,Z 879.132,A -85,B 0,C 180,E1 14882.28,E2 14882.28} C_VEL
LIN {X 0,Y 339.304,Z 1032.173,A -85,B 0,C 180,E1 14879.163,E2 14879.163} C_VEL
LIN {X 0,Y 338.737,Z 1051.361,A -85,B 0,C 180,E1 14878.601,E2 14878.601} C_VEL
LIN {X 0,Y 337.596,Z 1068.339,A -85,B 0,C 180,E1 14877.803,E2 14877.803} C_VEL
LIN {X 0,Y 335.851,Z 1084.814,A -85,B 0,C 180,E1 14876.712,E2 14876.712} C_VEL
LIN {X 0,Y 333.549,Z 1101.145,A -85,B 0,C 180,E1 14875.285,E2 14875.285} C_VEL
LIN {X 0,Y 331.063,Z 1115.531,A -85,B 0,C 180,E1 14873.681,E2 14873.681} C_VEL
LIN {X 0,Y 328.337,Z 1128.905,A -85,B 0,C 180,E1 14871.807,E2 14871.807} C_VEL
LIN {X 0,Y 325.409,Z 1141.736,A -85,B 0,C 180,E1 14869.565,E2 14869.565} C_VEL
LIN {X 0,Y 322.639,Z 1152.947,A -85,B 0,C 180,E1 14867.12,E2 14867.12} C_VEL
LIN {X 0,Y 320.13,Z 1162.538,A -85,B 0,C 180,E1 14864.467,E2 14864.467} C_VEL
LIN {X 0,Y 317.989,Z 1170.585,A -85,B 0,C 180,E1 14861.607,E2 14861.607} C_VEL
LIN {X 0,Y 316.31,Z 1177.074,A -85,B 0,C 180,E1 14858.542,E2 14858.542} C_VEL
LIN {X 0,Y 315.182,Z 1181.626,A -85,B 0,C 180,E1 14855.459,E2 14855.459} C_VEL
LIN {X 0,Y 314.522,Z 1184.528,A -85,B 0,C 180,E1 14852.184,E2 14852.184} C_VEL
LIN {X 0,Y 314.335,Z 1185.633,A -85,B 0,C 180,E1 14848.904,E2 14848.904} C_VEL
LIN {X 0,Y 314.587,Z 1184.931,A -85,B 0,C 180,E1 14845.623,E2 14845.623} C_VEL
LIN {X 0,Y 315.321,Z 1182.355,A -85,B 0,C 180,E1 14842.344,E2 14842.344} C_VEL
LIN {X 0,Y 316.558,Z 1178.109,A -85,B 0,C 180,E1 14839.216,E2 14839.216} C_VEL
LIN {X 0,Y 318.329,Z 1172.142,A -85,B 0,C 180,E1 14836.187,E2 14836.187} C_VEL
LIN {X 0,Y 320.574,Z 1164.468,A -85,B 0,C 180,E1 14833.322,E2 14833.322} C_VEL
LIN {X 0,Y 323.207,Z 1155.277,A -85,B 0,C 180,E1 14830.66,E2 14830.66} C_VEL
LIN {X 0,Y 326.099,Z 1144.666,A -85,B 0,C 180,E1 14828.22,E2 14828.22} C_VEL
LIN {X 0,Y 329.146,Z 1132.422,A -85,B 0,C 180,E1 14825.977,E2 14825.977} C_VEL
LIN {X 0,Y 332.11,Z 1119.047,A -85,B 0,C 180,E1 14824.018,E2 14824.018} C_VEL
LIN {X 0,Y 334.861,Z 1104.69,A -85,B 0,C 180,E1 14822.332,E2 14822.332} C_VEL
LIN {X 0,Y 337.294,Z 1089.346,A -85,B 0,C 180,E1 14820.909,E2 14820.909} C_VEL
LIN {X 0,Y 339.211,Z 1073.366,A -85,B 0,C 180,E1 14819.778,E2 14819.778} C_VEL
LIN {X 0,Y 340.657,Z 1055.613,A -85,B 0,C 180,E1 14818.863,E2 14818.863} C_VEL
LIN {X 0,Y 341.402,Z 1037.982,A -85,B 0,C 180,E1 14818.269,E2 14818.269} C_VEL
LIN {X 0,Y 343.21,Z 981.932,A -85,B 0,C 180,E1 14817.09,E2 14817.09} C_VEL
LIN {X 0,Y 347.395,Z 876.706,A -85,B 0,C 180,E1 14814.966,E2 14814.966} C_VEL
LIN {X 0,Y 346.962,Z 871.504,A -85,B 0,C 180,E1 14814.752,E2 14814.752} C_VEL
LIN {X 0,Y 347.326,Z 868.78,A -85,B 0,C 180,E1 14814.491,E2 14814.491} C_VEL
LIN {X 0,Y 348.905,Z 869.177,A -85,B 0,C 180,E1 14814.222,E2 14814.222} C_VEL
LIN {X 0,Y 351.764,Z 867.858,A -85,B 0,C 180,E1 14813.854,E2 14813.854} C_VEL
LIN {X 0,Y 355.757,Z 863.857,A -85,B 0,C 180,E1 14813.47,E2 14813.47} C_VEL
LIN {X 0,Y 356.975,Z 862.28,A -85,B 0,C 180,E1 14813.37,E2 14813.37} C_VEL
LIN {X 0,Y 361.043,Z 860.414,A -85,B 0,C 180,E1 14812.86,E2 14812.86} C_VEL
LIN {X 0,Y 365.66,Z 856.287,A -85,B 0,C 180,E1 14812.399,E2 14812.399} C_VEL
LIN {X 0,Y 367.387,Z 854.553,A -85,B 0,C 180,E1 14812.237,E2 14812.237} C_VEL
LIN {X 0,Y 372.429,Z 851.466,A -85,B 0,C 180,E1 14811.668,E2 14811.668} C_VEL
LIN {X 0,Y 377.793,Z 846.619,A -85,B 0,C 180,E1 14811.15,E2 14811.15} C_VEL
